C07280=1094.972,417.222,400.209,178.802,23.550,153.433
C07281=1094.966,417.006,400.244,178.799,23.542,153.431
C07282=1094.960,416.791,400.280,178.797,23.534,153.429
C07283=1094.956,416.575,400.315,178.794,23.526,153.428
C07284=1094.950,416.359,400.351,178.792,23.518,153.426
C07285=1094.945,416.144,400.387,178.789,23.510,153.424
C07286=1094.938,415.897,400.427,178.786,23.501,153.423
C07287=1094.933,415.650,400.467,178.783,23.492,153.421
C07288=1094.926,415.404,400.508,178.780,23.483,153.419
C07289=1094.920,415.157,400.548,178.778,23.475,153.417
C07290=1094.914,414.910,400.589,178.776,23.466,153.415
C07291=1094.908,414.664,400.629,178.772,23.457,153.414
C07292=1094.902,414.417,400.669,178.770,23.448,153.412
C07293=1094.896,414.170,400.710,178.767,23.439,153.410
C07294=1094.890,413.923,400.749,178.764,23.431,153.408
C07295=1094.883,413.677,400.789,178.762,23.422,153.407
C07296=1094.877,413.430,400.829,178.758,23.414,153.405
C07297=1094.871,413.184,400.870,178.756,23.405,153.403
C07298=1094.865,412.937,400.910,178.753,23.396,153.401
C07299=1094.859,412.690,400.950,178.750,23.387,153.400
C07300=1094.853,412.443,400.990,178.747,23.379,153.398
C07301=1094.847,412.197,401.030,178.744,23.371,153.396
C07302=1094.841,411.951,401.070,178.741,23.362,153.395
C07303=1094.835,411.704,401.110,178.738,23.353,153.393
C07304=1094.829,411.457,401.150,178.736,23.345,153.391
C07305=1094.823,411.210,401.191,178.733,23.337,153.390
C07306=1094.816,410.955,401.232,178.730,23.328,153.388
C07307=1094.810,410.698,401.273,178.727,23.319,153.386
C07308=1094.804,410.442,401.314,178.724,23.311,153.384
C07309=1094.798,410.186,401.356,178.721,23.302,153.383
C07310=1094.791,409.939,401.396,178.719,23.294,153.381
C07311=1094.785,409.692,401.435,178.716,23.286,153.379
C07312=1094.780,409.446,401.476,178.713,23.277,153.378
C07313=1094.774,409.199,401.515,178.711,23.269,153.376
C07314=1094.768,408.952,401.555,178.708,23.261,153.374
C07315=1094.762,408.705,401.595,178.705,23.253,153.373
C07316=1094.755,408.459,401.635,178.702,23.245,153.371
C07317=1094.750,408.212,401.674,178.699,23.237,153.370
C07318=1094.744,407.965,401.713,178.696,23.228,153.368
C07319=1094.738,407.718,401.754,178.694,23.220,153.366
C07320=1094.732,407.471,401.793,178.691,23.212,153.365
C07321=1094.727,407.225,401.833,178.688,23.205,153.363
C07322=1094.720,406.978,401.873,178.685,23.196,153.362
C07323=1094.714,406.731,401.912,178.682,23.188,153.360
C07324=1094.708,406.484,401.952,178.680,23.180,153.359
C07325=1094.703,406.237,401.991,178.677,23.172,153.357
C07326=1094.695,405.991,402.030,178.674,23.164,153.356
C07327=1094.689,405.744,402.070,178.671,23.156,153.354
C07328=1094.683,405.497,402.109,178.669,23.149,153.353
C07329=1094.678,405.250,402.148,178.666,23.141,153.351
C07330=1094.672,405.003,402.188,178.663,23.133,153.349
C07331=1094.666,404.756,402.227,178.660,23.126,153.348
C07332=1094.660,404.510,402.266,178.657,23.118,153.347
C07333=1094.654,404.263,402.305,178.655,23.110,153.345
C07334=1094.648,404.015,402.345,178.651,23.102,153.344
C07335=1094.642,403.769,402.383,178.649,23.095,153.342
C07336=1094.636,403.522,402.423,178.646,23.087,153.341
C07337=1094.630,403.275,402.462,178.643,23.080,153.339
C07338=1094.624,403.029,402.501,178.640,23.072,153.338
C07339=1094.617,402.782,402.540,178.638,23.064,153.336
C07340=1094.611,402.535,402.580,178.635,23.057,153.335
C07341=1094.606,402.288,402.619,178.632,23.049,153.333
C07342=1094.600,402.041,402.658,178.630,23.042,153.332
C07343=1094.593,401.794,402.697,178.626,23.034,153.331
C07344=1094.588,401.548,402.736,178.624,23.027,153.329
C07345=1094.581,401.301,402.775,178.620,23.019,153.328
C07346=1094.576,401.054,402.814,178.618,23.012,153.326
C07347=1094.569,400.807,402.853,178.615,23.005,153.325
C07348=1094.564,400.560,402.892,178.612,22.997,153.324
C07349=1094.558,400.313,402.931,178.610,22.990,153.322
C07350=1094.551,400.066,402.969,178.607,22.982,153.321
C07351=1094.546,399.819,403.008,178.604,22.975,153.319
C07352=1094.540,399.572,403.048,178.601,22.968,153.318
C07353=1094.534,399.326,403.085,178.598,22.961,153.317
C07354=1094.528,399.078,403.125,178.596,22.954,153.315
C07355=1094.522,398.832,403.163,178.592,22.946,153.314
C07356=1094.516,398.584,403.202,178.590,22.939,153.313
C07357=1094.510,398.338,403.241,178.587,22.932,153.311
C07358=1094.504,398.118,403.275,178.585,22.926,153.310
C07359=1094.499,397.898,403.309,178.582,22.919,153.309
C07360=1094.493,397.677,403.344,178.579,22.913,153.308
C07361=1094.489,397.458,403.379,178.577,22.907,153.306
C07362=1094.483,397.237,403.414,178.575,22.900,153.305
C07363=1094.478,397.017,403.448,178.572,22.894,153.304
C07364=1094.473,396.798,403.482,178.569,22.888,153.303
C07365=1094.468,396.577,403.516,178.567,22.882,153.302
C07366=1094.461,396.331,403.555,178.564,22.874,153.301
C07367=1094.455,396.083,403.593,178.561,22.868,153.299
C07368=1094.450,395.836,403.631,178.559,22.861,153.298
C07369=1094.443,395.590,403.670,178.556,22.854,153.297
C07370=1094.438,395.343,403.708,178.553,22.847,153.295
C07371=1094.432,395.096,403.746,178.550,22.840,153.294
C07372=1094.426,394.849,403.786,178.548,22.833,153.293
C07373=1094.420,394.602,403.823,178.544,22.826,153.292
C07374=1094.414,394.355,403.861,178.541,22.819,153.290
C07375=1094.408,394.108,403.901,178.539,22.813,153.289
C07376=1094.402,393.861,403.938,178.536,22.806,153.288
C07377=1094.396,393.615,403.976,178.533,22.799,153.287
C07378=1094.390,393.367,404.015,178.530,22.792,153.285
C07379=1094.384,393.121,404.053,178.527,22.786,153.284
C07380=1094.378,392.874,404.091,178.525,22.779,153.283
C07381=1094.372,392.626,404.129,178.521,22.772,153.282
C07382=1094.366,392.379,404.167,178.519,22.765,153.281
C07383=1094.361,392.133,404.205,178.516,22.759,153.279
C07384=1094.354,391.885,404.243,178.513,22.752,153.278
C07385=1094.348,391.638,404.281,178.511,22.746,153.277
C07386=1094.342,391.392,404.319,178.507,22.739,153.276
C07387=1094.336,391.144,404.357,178.504,22.732,153.275
C07388=1094.330,390.898,404.395,178.502,22.726,153.274
C07389=1094.324,390.651,404.434,178.499,22.720,153.272
C07390=1094.318,390.403,404.471,178.496,22.713,153.271
C07391=1094.312,390.156,404.509,178.493,22.706,153.270
C07392=1094.306,389.910,404.547,178.490,22.700,153.269
C07393=1094.300,389.663,404.584,178.487,22.694,153.268
C07394=1094.295,389.416,404.622,178.485,22.687,153.267
C07395=1094.288,389.169,404.660,178.482,22.681,153.266
C07396=1094.282,388.922,404.698,178.478,22.674,153.265
C07397=1094.276,388.675,404.736,178.475,22.668,153.263
C07398=1094.270,388.428,404.774,178.473,22.662,153.262
C07399=1094.264,388.182,404.811,178.470,22.655,153.261
C07400=1094.258,387.934,404.849,178.467,22.649,153.260
C07401=1094.252,387.687,404.887,178.464,22.643,153.259
C07402=1094.246,387.440,404.924,178.461,22.636,153.258
C07403=1094.240,387.193,404.962,178.458,22.630,153.257
C07404=1094.235,386.947,405.000,178.455,22.624,153.256
C07405=1094.229,386.699,405.037,178.452,22.617,153.254
C07406=1094.223,386.453,405.075,178.450,22.611,153.253
C07407=1094.217,386.205,405.113,178.447,22.605,153.252
C07408=1094.211,385.958,405.150,178.444,22.599,153.251
C07409=1094.205,385.711,405.188,178.441,22.593,153.250
C07410=1094.199,385.464,405.225,178.438,22.586,153.249
C07411=1094.194,385.217,405.262,178.435,22.580,153.248
C07412=1094.188,384.970,405.300,178.432,22.574,153.247
C07413=1094.182,384.723,405.337,178.429,22.568,153.246
C07414=1094.177,384.509,405.370,178.427,22.563,153.245
C07415=1094.172,384.296,405.402,178.424,22.557,153.244
C07416=1094.166,384.082,405.434,178.422,22.552,153.243
C07417=1094.161,383.869,405.466,178.420,22.547,153.242
C07418=1094.156,383.655,405.498,178.417,22.542,153.242
C07419=1094.151,383.441,405.531,178.415,22.536,153.240
C07420=1094.146,383.228,405.563,178.411,22.531,153.240
C07421=1094.142,383.014,405.595,178.409,22.525,153.239
C07422=1094.136,382.767,405.633,178.406,22.519,153.238
C07423=1094.130,382.520,405.670,178.404,22.514,153.237
C07424=1094.124,382.273,405.706,178.401,22.508,153.236
C07425=1094.118,382.026,405.744,178.398,22.502,153.235
C07426=1094.112,381.778,405.782,178.395,22.496,153.234
C07427=1094.105,381.531,405.818,178.392,22.490,153.233
C07428=1094.099,381.284,405.856,178.389,22.485,153.232
C07429=1094.094,381.037,405.893,178.386,22.479,153.231
C07430=1094.087,380.790,405.929,178.383,22.473,153.230
C07431=1094.081,380.543,405.967,178.380,22.467,153.229
C07432=1094.076,380.296,406.004,178.377,22.461,153.228
C07433=1094.070,380.049,406.041,178.374,22.455,153.227
C07434=1094.064,379.801,406.078,178.371,22.450,153.226
C07435=1094.058,379.554,406.115,178.369,22.444,153.225
C07436=1094.052,379.308,406.151,178.366,22.438,153.224
C07437=1094.047,379.061,406.188,178.363,22.432,153.223
C07438=1094.040,378.814,406.225,178.360,22.427,153.222
C07439=1094.035,378.567,406.262,178.357,22.421,153.221
C07440=1094.029,378.319,406.299,178.354,22.415,153.220
C07441=1094.023,378.072,406.335,178.351,22.409,153.220
C07442=1094.017,377.825,406.372,178.348,22.403,153.218
C07443=1094.011,377.578,406.409,178.345,22.398,153.218
C07444=1094.005,377.330,406.446,178.342,22.392,153.217
C07445=1093.999,377.083,406.482,178.339,22.386,153.216
C07446=1093.993,376.836,406.519,178.336,22.381,153.215
C07447=1093.988,376.589,406.556,178.333,22.375,153.214
C07448=1093.982,376.342,406.593,178.330,22.370,153.213
C07449=1093.976,376.095,406.630,178.327,22.364,153.212
C07450=1093.970,375.848,406.666,178.324,22.358,153.211
C07451=1093.965,375.600,406.703,178.321,22.353,153.210
C07452=1093.958,375.353,406.739,178.318,22.347,153.209
C07453=1093.953,375.105,406.776,178.315,22.342,153.209
C07454=1093.947,374.859,406.812,178.312,22.336,153.208
C07455=1093.942,374.612,406.849,178.309,22.331,153.207
C07456=1093.935,374.365,406.885,178.307,22.325,153.206
C07457=1093.930,374.117,406.922,178.304,22.320,153.205
C07458=1093.924,373.870,406.958,178.301,22.314,153.204
C07459=1093.917,373.623,406.995,178.298,22.309,153.203
C07460=1093.912,373.376,407.031,178.295,22.304,153.203
C07461=1093.906,373.129,407.068,178.292,22.298,153.202
C07462=1093.900,372.881,407.103,178.289,22.293,153.201
C07463=1093.894,372.634,407.140,178.285,22.287,153.200
C07464=1093.888,372.387,407.177,178.282,22.282,153.199
C07465=1093.883,372.140,407.212,178.280,22.277,153.198
C07466=1093.876,371.893,407.249,178.277,22.272,153.198
C07467=1093.871,371.645,407.285,178.274,22.266,153.197
C07468=1093.865,371.398,407.322,178.271,22.261,153.196
C07469=1093.858,371.151,407.358,178.268,22.255,153.195
C07470=1093.849,370.751,407.416,178.263,22.247,153.194
C07471=1093.840,370.351,407.474,178.258,22.238,153.192
C07472=1093.830,369.951,407.533,178.254,22.230,153.191
C07473=1093.821,369.552,407.591,178.249,22.222,153.190
C07474=1093.815,369.304,407.627,178.246,22.217,153.189
C07475=1093.808,369.057,407.663,178.243,22.211,153.188
C07476=1093.804,368.810,407.699,178.240,22.206,153.187
C07477=1093.798,368.562,407.735,178.236,22.201,153.187
C07478=1093.791,368.315,407.771,178.234,22.196,153.186
C07479=1093.785,368.067,407.807,178.231,22.190,153.185
C07480=1093.780,367.820,407.843,178.228,22.185,153.184
C07481=1093.774,367.573,407.880,178.225,22.180,153.184
C07482=1093.769,367.326,407.915,178.222,22.175,153.183
C07483=1093.763,367.078,407.951,178.218,22.170,153.182
C07484=1093.757,366.831,407.986,178.216,22.165,153.181
C07485=1093.751,366.584,408.023,178.213,22.160,153.180
C07486=1093.745,366.337,408.058,178.210,22.155,153.180
C07487=1093.739,366.089,408.094,178.207,22.150,153.179
C07488=1093.734,365.842,408.129,178.204,22.144,153.178
C07489=1093.728,365.594,408.165,178.201,22.140,153.177
C07490=1093.722,365.347,408.201,178.198,22.135,153.177
C07491=1093.716,365.100,408.237,178.195,22.130,153.176
C07492=1093.710,364.853,408.273,178.192,22.125,153.175
C07493=1093.704,364.606,408.308,178.189,22.120,153.175
C07494=1093.698,364.358,408.344,178.186,22.115,153.174
C07495=1093.692,364.110,408.379,178.183,22.110,153.173
C07496=1093.687,363.863,408.415,178.180,22.105,153.172
C07497=1093.681,363.616,408.451,178.177,22.101,153.172
C07498=1093.675,363.369,408.486,178.174,22.095,153.171
C07499=1093.669,363.121,408.522,178.171,22.090,153.170
C07500=1093.663,362.873,408.557,178.168,22.085,153.170
C07501=1093.658,362.626,408.593,178.165,22.081,153.169
C07502=1093.652,362.379,408.628,178.162,22.076,153.168
C07503=1093.647,362.132,408.664,178.159,22.071,153.168
C07504=1093.640,361.884,408.699,178.156,22.066,153.167
C07505=1093.635,361.637,408.734,178.153,22.061,153.166
C07506=1093.629,361.389,408.769,178.150,22.057,153.166
C07507=1093.623,361.141,408.805,178.147,22.052,153.165
C07508=1093.617,360.894,408.840,178.143,22.047,153.164
C07509=1093.611,360.647,408.876,178.141,22.042,153.163
C07510=1093.605,360.400,408.911,178.138,22.038,153.163
C07511=1093.599,360.152,408.946,178.135,22.032,153.162
C07512=1093.594,359.905,408.981,178.132,22.028,153.161
C07513=1093.588,359.657,409.017,178.129,22.024,153.161
C07514=1093.583,359.409,409.052,178.126,22.018,153.160
C07515=1093.576,359.162,409.087,178.122,22.014,153.160
C07516=1093.570,358.915,409.122,178.120,22.009,153.159
C07517=1093.564,358.667,409.158,178.117,22.004,153.158
C07518=1093.559,358.420,409.192,178.113,22.000,153.158
C07519=1093.553,358.172,409.228,178.111,21.995,153.157
C07520=1093.547,357.925,409.262,178.107,21.991,153.156
C07521=1093.541,357.678,409.297,178.104,21.986,153.156
C07522=1093.532,357.293,409.351,178.100,21.979,153.155
C07523=1093.523,356.908,409.407,178.095,21.972,153.154
C07524=1093.514,356.524,409.461,178.091,21.965,153.153
C07525=1093.505,356.139,409.515,178.085,21.957,153.152
C07526=1093.499,355.892,409.550,178.083,21.953,153.151
C07527=1093.493,355.644,409.585,178.080,21.948,153.151
C07528=1093.488,355.397,409.620,178.076,21.943,153.150
C07529=1093.482,355.150,409.654,178.074,21.939,153.149
C07530=1093.476,354.902,409.690,178.070,21.934,153.149
C07531=1093.470,354.655,409.724,178.067,21.930,153.148
C07532=1093.464,354.406,409.759,178.065,21.926,153.147
C07533=1093.459,354.160,409.794,178.061,21.921,153.147
C07534=1093.453,353.912,409.828,178.059,21.917,153.146
C07535=1093.447,353.664,409.863,178.055,21.912,153.146
C07536=1093.441,353.417,409.898,178.052,21.908,153.145
C07537=1093.436,353.170,409.933,178.049,21.903,153.145
C07538=1093.430,352.922,409.967,178.046,21.899,153.144
C07539=1093.425,352.674,410.002,178.043,21.894,153.143
C07540=1093.418,352.427,410.037,178.040,21.890,153.143
C07541=1093.412,352.179,410.071,178.037,21.886,153.142
C07542=1093.407,351.932,410.106,178.034,21.881,153.142
C07543=1093.400,351.684,410.140,178.031,21.877,153.141
C07544=1093.395,351.436,410.175,178.027,21.872,153.141
C07545=1093.389,351.190,410.209,178.025,21.868,153.140
C07546=1093.383,350.942,410.244,178.021,21.864,153.140
C07547=1093.377,350.694,410.279,178.019,21.860,153.139
C07548=1093.372,350.447,410.313,178.016,21.855,153.138
C07549=1093.367,350.199,410.347,178.012,21.851,153.138
C07550=1093.360,349.951,410.382,178.010,21.846,153.137
C07551=1093.354,349.704,410.416,178.006,21.842,153.137
C07552=1093.349,349.456,410.450,178.004,21.838,153.136
C07553=1093.343,349.208,410.485,178.000,21.834,153.136
C07554=1093.337,348.961,410.519,177.998,21.829,153.135
C07555=1093.332,348.713,410.553,177.994,21.825,153.135
C07556=1093.326,348.466,410.588,177.992,21.821,153.134
C07557=1093.319,348.218,410.622,177.988,21.817,153.134
C07558=1093.313,347.971,410.656,177.985,21.812,153.133
C07559=1093.308,347.723,410.691,177.982,21.808,153.133
C07560=1093.302,347.476,410.725,177.979,21.804,153.132
C07561=1093.296,347.228,410.759,177.976,21.800,153.131
C07562=1093.291,346.980,410.794,177.973,21.795,153.131
C07563=1093.285,346.733,410.827,177.970,21.791,153.130
C07564=1093.279,346.485,410.861,177.967,21.787,153.130
C07565=1093.274,346.238,410.895,177.964,21.783,153.129
C07566=1093.268,345.991,410.929,177.961,21.778,153.129
C07567=1093.262,345.742,410.964,177.958,21.775,153.128
C07568=1093.256,345.494,410.998,177.955,21.770,153.128
C07569=1093.251,345.247,411.032,177.951,21.766,153.127
C07570=1093.245,345.000,411.066,177.949,21.762,153.127
C07571=1093.239,344.753,411.100,177.945,21.758,153.126
C07572=1093.233,344.504,411.134,177.942,21.754,153.126
C07573=1093.228,344.256,411.168,177.939,21.750,153.125
C07574=1093.219,343.874,411.220,177.934,21.743,153.125
C07575=1093.209,343.492,411.273,177.930,21.737,153.124
C07576=1093.201,343.110,411.324,177.925,21.731,153.123
C07577=1093.191,342.728,411.377,177.921,21.725,153.123
C07578=1093.186,342.481,411.411,177.917,21.721,153.122
C07579=1093.180,342.233,411.445,177.914,21.717,153.122
C07580=1093.174,341.985,411.478,177.911,21.713,153.121
C07581=1093.168,341.738,411.512,177.908,21.709,153.121
C07582=1093.163,341.490,411.545,177.905,21.705,153.120
C07583=1093.157,341.243,411.579,177.902,21.701,153.120
C07584=1093.151,340.995,411.613,177.899,21.697,153.119
C07585=1093.146,340.748,411.647,177.896,21.693,153.119
C07586=1093.140,340.500,411.680,177.892,21.688,153.118
C07587=1093.134,340.252,411.715,177.890,21.685,153.118
C07588=1093.128,340.004,411.748,177.886,21.680,153.117
C07589=1093.122,339.756,411.781,177.883,21.677,153.117
C07590=1093.117,339.509,411.815,177.881,21.673,153.117
C07591=1093.111,339.261,411.849,177.877,21.669,153.116
C07592=1093.106,339.013,411.882,177.875,21.665,153.116
C07593=1093.100,338.766,411.916,177.871,21.661,153.115
C07594=1093.094,338.518,411.949,177.868,21.657,153.115
C07595=1093.088,338.270,411.982,177.865,21.653,153.114
C07596=1093.082,338.023,412.016,177.862,21.650,153.114
C07597=1093.076,337.775,412.050,177.859,21.646,153.113
C07598=1093.071,337.527,412.083,177.856,21.642,153.113
C07599=1093.065,337.279,412.116,177.853,21.638,153.113
C07600=1093.059,337.032,412.149,177.850,21.634,153.112
C07601=1093.053,336.784,412.183,177.847,21.630,153.112
C07602=1093.048,336.536,412.216,177.843,21.626,153.111
C07603=1093.042,336.288,412.250,177.840,21.623,153.111
C07604=1093.036,336.041,412.282,177.838,21.619,153.111
C07605=1093.030,335.793,412.316,177.834,21.615,153.110
C07606=1093.025,335.545,412.349,177.831,21.611,153.110
C07607=1093.019,335.298,412.383,177.828,21.607,153.109
C07608=1093.012,335.050,412.416,177.825,21.604,153.109
C07609=1093.007,334.802,412.449,177.822,21.600,153.109
C07610=1093.001,334.554,412.483,177.819,21.596,153.108
C07611=1092.996,334.306,412.516,177.816,21.592,153.108
C07612=1092.989,334.059,412.549,177.812,21.589,153.107
C07613=1092.984,333.811,412.582,177.810,21.585,153.107
C07614=1092.979,333.564,412.615,177.807,21.581,153.107
C07615=1092.973,333.316,412.648,177.803,21.577,153.106
C07616=1092.967,333.068,412.681,177.801,21.574,153.106
C07617=1092.962,332.820,412.714,177.798,21.570,153.105
C07618=1092.955,332.573,412.747,177.794,21.566,153.105
C07619=1092.950,332.324,412.780,177.792,21.562,153.105
C07620=1092.944,332.076,412.813,177.788,21.559,153.104
C07621=1092.938,331.829,412.846,177.785,21.555,153.104
C07622=1092.933,331.581,412.879,177.782,21.551,153.103
C07623=1092.926,331.333,412.912,177.779,21.548,153.103
C07624=1092.920,331.086,412.945,177.776,21.544,153.103
C07625=1092.915,330.838,412.978,177.773,21.541,153.103
C07626=1092.905,330.450,413.029,177.768,21.535,153.102
C07627=1092.896,330.062,413.080,177.763,21.529,153.101
C07628=1092.887,329.674,413.132,177.758,21.524,153.101
C07629=1092.878,329.286,413.183,177.754,21.518,153.100
C07630=1092.872,329.039,413.215,177.750,21.515,153.100
C07631=1092.867,328.790,413.248,177.747,21.511,153.100
C07632=1092.861,328.542,413.281,177.745,21.508,153.099
C07633=1092.854,328.295,413.314,177.741,21.504,153.099
C07634=1092.849,328.046,413.346,177.738,21.501,153.099
C07635=1092.843,327.799,413.379,177.735,21.497,153.098
C07636=1092.837,327.551,413.411,177.732,21.493,153.098
C07637=1092.832,327.303,413.444,177.729,21.490,153.098
C07638=1092.826,327.056,413.477,177.726,21.487,153.097
C07639=1092.820,326.808,413.509,177.722,21.482,153.097
C07640=1092.815,326.560,413.542,177.720,21.479,153.097
C07641=1092.809,326.312,413.574,177.717,21.476,153.096
C07642=1092.802,326.065,413.606,177.714,21.472,153.096
C07643=1092.797,325.816,413.639,177.710,21.469,153.096
C07644=1092.791,325.569,413.671,177.707,21.465,153.095
C07645=1092.785,325.321,413.703,177.705,21.462,153.095
C07646=1092.780,325.073,413.737,177.701,21.458,153.095
C07647=1092.774,324.825,413.769,177.698,21.455,153.094
C07648=1092.768,324.578,413.801,177.695,21.452,153.094
C07649=1092.762,324.330,413.833,177.692,21.448,153.094
C07650=1092.757,324.081,413.866,177.688,21.445,153.093
C07651=1092.751,323.834,413.899,177.686,21.441,153.093
C07652=1092.745,323.586,413.930,177.683,21.438,153.093
C07653=1092.739,323.338,413.963,177.680,21.435,153.092
C07654=1092.734,323.090,413.996,177.676,21.431,153.092
C07655=1092.728,322.842,414.027,177.673,21.427,153.092
C07656=1092.722,322.594,414.059,177.671,21.424,153.091
C07657=1092.716,322.347,414.092,177.668,21.421,153.091
C07658=1092.711,322.099,414.124,177.664,21.417,153.091
C07659=1092.705,321.851,414.156,177.661,21.414,153.091
C07660=1092.700,321.604,414.189,177.658,21.410,153.090
C07661=1092.694,321.355,414.221,177.655,21.407,153.090
C07662=1092.688,321.107,414.253,177.652,21.403,153.090
C07663=1092.682,320.860,414.284,177.649,21.400,153.089
C07664=1092.677,320.611,414.317,177.646,21.397,153.089
C07665=1092.671,320.364,414.350,177.643,21.394,153.089
C07666=1092.665,320.116,414.381,177.639,21.390,153.089
C07667=1092.659,319.868,414.413,177.637,21.386,153.088
C07668=1092.654,319.620,414.445,177.634,21.383,153.088
C07669=1092.648,319.372,414.477,177.631,21.380,153.088
C07670=1092.643,319.124,414.509,177.627,21.376,153.087
C07671=1092.637,318.876,414.541,177.624,21.373,153.087
C07672=1092.632,318.629,414.573,177.621,21.370,153.087
C07673=1092.626,318.380,414.605,177.619,21.366,153.086
C07674=1092.621,318.133,414.637,177.616,21.363,153.086
C07675=1092.615,317.885,414.669,177.612,21.360,153.086
C07676=1092.609,317.637,414.700,177.609,21.356,153.086
C07677=1092.603,317.389,414.733,177.606,21.353,153.085
C07678=1092.595,316.994,414.784,177.601,21.347,153.085
C07679=1092.586,316.599,414.835,177.597,21.343,153.084
C07680=1092.577,316.204,414.885,177.592,21.337,153.084
C07681=1092.568,315.809,414.935,177.587,21.332,153.083
C07682=1092.563,315.562,414.968,177.584,21.328,153.083
C07683=1092.557,315.313,415.000,177.581,21.325,153.083
C07684=1092.552,315.066,415.031,177.578,21.322,153.083
C07685=1092.545,314.818,415.063,177.574,21.319,153.082
C07686=1092.540,314.570,415.094,177.571,21.315,153.082
C07687=1092.534,314.322,415.126,177.568,21.312,153.082
C07688=1092.527,314.074,415.157,177.565,21.309,153.082
C07689=1092.522,313.826,415.189,177.562,21.306,153.081
C07690=1092.516,313.578,415.221,177.559,21.303,153.081
C07691=1092.511,313.330,415.252,177.556,21.299,153.081
C07692=1092.504,313.082,415.283,177.553,21.296,153.081
C07693=1092.499,312.834,415.315,177.550,21.293,153.081
C07694=1092.493,312.586,415.347,177.547,21.290,153.080
C07695=1092.487,312.338,415.377,177.544,21.287,153.080
C07696=1092.481,312.091,415.409,177.541,21.284,153.080
C07697=1092.475,311.843,415.441,177.537,21.281,153.080
C07698=1092.470,311.595,415.471,177.534,21.277,153.079
C07699=1092.464,311.347,415.503,177.531,21.275,153.079
C07700=1092.458,311.099,415.534,177.528,21.272,153.079
C07701=1092.452,310.851,415.566,177.525,21.268,153.079
C07702=1092.446,310.603,415.597,177.522,21.265,153.078
C07703=1092.441,310.355,415.628,177.519,21.262,153.078
C07704=1092.435,310.107,415.660,177.515,21.259,153.078
C07705=1092.429,309.859,415.691,177.513,21.256,153.078
C07706=1092.423,309.611,415.722,177.509,21.253,153.078
C07707=1092.418,309.363,415.753,177.506,21.250,153.077
C07708=1092.412,309.115,415.785,177.503,21.247,153.077
C07709=1092.406,308.867,415.815,177.501,21.244,153.077
C07710=1092.400,308.619,415.847,177.498,21.241,153.077
C07711=1092.395,308.372,415.877,177.494,21.237,153.077
C07712=1092.389,308.123,415.909,177.491,21.234,153.076
C07713=1092.383,307.875,415.940,177.488,21.231,153.076
C07714=1092.377,307.628,415.972,177.485,21.228,153.076
C07715=1092.372,307.379,416.003,177.482,21.225,153.076
C07716=1092.366,307.132,416.034,177.479,21.222,153.075
C07717=1092.361,306.884,416.065,177.476,21.219,153.075
C07718=1092.354,306.635,416.096,177.472,21.216,153.075
C07719=1092.349,306.388,416.127,177.469,21.213,153.075
C07720=1092.343,306.140,416.158,177.466,21.210,153.075
C07721=1092.338,305.892,416.189,177.463,21.207,153.074
C07722=1092.331,305.644,416.220,177.460,21.204,153.074
C07723=1092.326,305.396,416.251,177.457,21.201,153.074
C07724=1092.320,305.148,416.281,177.454,21.198,153.074
C07725=1092.315,304.900,416.312,177.451,21.195,153.074
C07726=1092.309,304.653,416.343,177.447,21.191,153.073
C07727=1092.303,304.404,416.375,177.444,21.188,153.073
C07728=1092.298,304.156,416.405,177.441,21.185,153.073
C07729=1092.292,303.908,416.436,177.438,21.183,153.073
C07730=1092.283,303.516,416.485,177.434,21.178,153.072
C07731=1092.274,303.123,416.533,177.429,21.173,153.072
C07732=1092.265,302.732,416.582,177.424,21.168,153.072
C07733=1092.257,302.339,416.631,177.419,21.163,153.072
C07734=1092.251,302.091,416.661,177.416,21.160,153.071
C07735=1092.246,301.843,416.692,177.413,21.157,153.071
C07736=1092.240,301.595,416.723,177.410,21.154,153.071
C07737=1092.234,301.347,416.753,177.407,21.151,153.071
C07738=1092.229,301.099,416.784,177.404,21.149,153.071
C07739=1092.223,300.851,416.814,177.401,21.146,153.070
C07740=1092.218,300.603,416.845,177.398,21.143,153.070
C07741=1092.212,300.355,416.876,177.395,21.140,153.070
C07742=1092.206,300.107,416.906,177.391,21.136,153.070
C07743=1092.201,299.858,416.937,177.388,21.133,153.070
C07744=1092.195,299.611,416.968,177.385,21.130,153.069
C07745=1092.189,299.363,416.998,177.382,21.127,153.069
C07746=1092.184,299.115,417.029,177.379,21.124,153.069
C07747=1092.178,298.867,417.059,177.376,21.121,153.069
C07748=1092.173,298.619,417.090,177.373,21.118,153.069
C07749=1092.167,298.371,417.121,177.370,21.115,153.068
C07750=1092.161,298.123,417.151,177.367,21.113,153.068
C07751=1092.156,297.875,417.181,177.364,21.110,153.068
C07752=1092.151,297.627,417.211,177.361,21.107,153.068
C07753=1092.145,297.379,417.242,177.358,21.104,153.068
C07754=1092.139,297.131,417.272,177.355,21.101,153.068
C07755=1092.133,296.883,417.303,177.352,21.098,153.068
C07756=1092.127,296.634,417.333,177.349,21.096,153.067
C07757=1092.121,296.386,417.363,177.346,21.093,153.067
C07758=1092.116,296.138,417.393,177.343,21.090,153.067
C07759=1092.111,295.890,417.424,177.340,21.087,153.067
C07760=1092.105,295.642,417.454,177.337,21.084,153.067
C07761=1092.099,295.394,417.484,177.334,21.081,153.067
C07762=1092.093,295.146,417.515,177.331,21.078,153.066
C07763=1092.088,294.898,417.544,177.328,21.076,153.066
C07764=1092.082,294.650,417.575,177.325,21.073,153.066
C07765=1092.076,294.402,417.605,177.321,21.070,153.066
C07766=1092.071,294.154,417.634,177.318,21.067,153.066
C07767=1092.065,293.906,417.665,177.315,21.064,153.066
C07768=1092.059,293.658,417.695,177.312,21.061,153.065
C07769=1092.054,293.409,417.725,177.309,21.058,153.065
C07770=1092.048,293.162,417.755,177.305,21.056,153.065
C07771=1092.042,292.913,417.785,177.302,21.053,153.065
C07772=1092.036,292.665,417.815,177.299,21.050,153.065
C07773=1092.031,292.417,417.845,177.296,21.047,153.065
C07774=1092.025,292.169,417.875,177.293,21.044,153.065
C07775=1092.020,291.921,417.905,177.290,21.041,153.065
C07776=1092.014,291.673,417.935,177.287,21.038,153.064
C07777=1092.008,291.424,417.965,177.284,21.036,153.064
C07778=1092.003,291.177,417.995,177.281,21.033,153.064
C07779=1091.997,290.928,418.025,177.278,21.030,153.064
C07780=1091.991,290.680,418.054,177.275,21.027,153.064
C07781=1091.985,290.432,418.084,177.272,21.025,153.064
C07782=1091.977,290.054,418.130,177.267,21.020,153.063
C07783=1091.969,289.675,418.175,177.262,21.016,153.063
C07784=1091.960,289.297,418.221,177.258,21.012,153.063
C07785=1091.951,288.919,418.266,177.253,21.008,153.063
C07786=1091.945,288.671,418.295,177.250,21.005,153.063
C07787=1091.939,288.423,418.325,177.247,21.003,153.063
C07788=1091.934,288.175,418.355,177.244,21.000,153.063
C07789=1091.928,287.926,418.385,177.241,20.997,153.062
C07790=1091.922,287.678,418.414,177.238,20.994,153.062
C07791=1091.917,287.431,418.444,177.235,20.992,153.062
C07792=1091.911,287.182,418.473,177.232,20.989,153.062
C07793=1091.906,286.934,418.503,177.229,20.986,153.062
C07794=1091.899,286.686,418.532,177.226,20.984,153.062
C07795=1091.894,286.437,418.562,177.223,20.981,153.062
C07796=1091.888,286.190,418.592,177.220,20.979,153.062
C07797=1091.882,285.941,418.621,177.217,20.976,153.061
C07798=1091.876,285.693,418.651,177.214,20.973,153.061
C07799=1091.871,285.445,418.680,177.211,20.970,153.061
C07800=1091.866,285.197,418.710,177.208,20.968,153.061
C07801=1091.860,284.949,418.739,177.204,20.965,153.061
C07802=1091.854,284.700,418.768,177.202,20.962,153.061
C07803=1091.849,284.452,418.798,177.198,20.960,153.061
C07804=1091.842,284.204,418.827,177.195,20.957,153.061
C07805=1091.837,283.956,418.856,177.192,20.954,153.061
C07806=1091.832,283.707,418.886,177.189,20.951,153.060
C07807=1091.826,283.459,418.915,177.186,20.948,153.060
C07808=1091.820,283.211,418.945,177.183,20.946,153.060
C07809=1091.815,282.963,418.974,177.180,20.943,153.060
C07810=1091.809,282.715,419.003,177.177,20.941,153.060
C07811=1091.803,282.467,419.032,177.175,20.938,153.060
C07812=1091.798,282.218,419.062,177.171,20.936,153.060
C07813=1091.792,281.971,419.091,177.168,20.933,153.060
C07814=1091.787,281.722,419.120,177.165,20.930,153.060
C07815=1091.780,281.474,419.149,177.162,20.927,153.059
C07816=1091.775,281.226,419.179,177.159,20.925,153.059
C07817=1091.770,280.978,419.208,177.156,20.922,153.059
C07818=1091.764,280.729,419.237,177.153,20.919,153.059
C07819=1091.758,280.481,419.266,177.149,20.917,153.059
C07820=1091.752,280.233,419.295,177.146,20.914,153.059
C07821=1091.747,279.985,419.324,177.143,20.912,153.059
C07822=1091.741,279.737,419.354,177.140,20.909,153.059
C07823=1091.735,279.488,419.382,177.138,20.907,153.059
C07824=1091.730,279.240,419.412,177.135,20.904,153.059
C07825=1091.724,278.992,419.440,177.132,20.901,153.058
C07826=1091.719,278.744,419.470,177.128,20.899,153.058
C07827=1091.713,278.495,419.498,177.125,20.896,153.058
C07828=1091.707,278.246,419.528,177.122,20.893,153.058
C07829=1091.701,277.999,419.557,177.119,20.891,153.058
C07830=1091.696,277.750,419.585,177.116,20.888,153.058
C07831=1091.690,277.502,419.615,177.113,20.886,153.058
C07832=1091.684,277.254,419.643,177.111,20.883,153.058
C07833=1091.679,277.005,419.672,177.108,20.881,153.058
C07834=1091.670,276.637,419.715,177.103,20.877,153.058
C07835=1091.662,276.268,419.758,177.098,20.873,153.058
C07836=1091.654,275.899,419.801,177.093,20.869,153.057
C07837=1091.646,275.530,419.843,177.090,20.865,153.057
C07838=1091.639,275.282,419.872,177.086,20.863,153.057
C07839=1091.634,275.034,419.900,177.083,20.860,153.057
C07840=1091.628,274.786,419.929,177.080,20.858,153.057
C07841=1091.623,274.537,419.958,177.077,20.855,153.057
C07842=1091.617,274.289,419.987,177.074,20.852,153.057
C07843=1091.611,274.040,420.015,177.071,20.850,153.057
C07844=1091.606,273.793,420.045,177.068,20.847,153.057
C07845=1091.600,273.544,420.073,177.065,20.845,153.057
C07846=1091.594,273.296,420.102,177.062,20.842,153.057
C07847=1091.589,273.048,420.130,177.059,20.840,153.056
C07848=1091.583,272.799,420.160,177.056,20.837,153.056
C07849=1091.578,272.551,420.188,177.053,20.834,153.056
C07850=1091.572,272.302,420.216,177.050,20.832,153.056
C07851=1091.566,272.054,420.245,177.046,20.830,153.056
C07852=1091.560,271.806,420.273,177.044,20.828,153.056
C07853=1091.554,271.558,420.301,177.041,20.825,153.056
C07854=1091.549,271.310,420.330,177.038,20.822,153.056
C07855=1091.543,271.061,420.359,177.035,20.820,153.056
C07856=1091.538,270.813,420.387,177.032,20.817,153.056
C07857=1091.532,270.564,420.415,177.028,20.814,153.056
C07858=1091.527,270.317,420.444,177.026,20.812,153.056
C07859=1091.521,270.068,420.472,177.023,20.810,153.056
C07860=1091.515,269.820,420.500,177.020,20.807,153.056
C07861=1091.510,269.571,420.529,177.017,20.804,153.055
C07862=1091.504,269.323,420.558,177.013,20.802,153.055
C07863=1091.498,269.075,420.586,177.010,20.800,153.055
C07864=1091.492,268.826,420.614,177.008,20.798,153.055
C07865=1091.487,268.578,420.642,177.005,20.795,153.055
C07866=1091.481,268.329,420.671,177.002,20.792,153.055
C07867=1091.476,268.081,420.699,176.998,20.790,153.055
C07868=1091.470,267.832,420.727,176.995,20.787,153.055
C07869=1091.464,267.585,420.756,176.992,20.785,153.055
C07870=1091.458,267.336,420.784,176.990,20.783,153.055
C07871=1091.453,267.088,420.812,176.987,20.780,153.055
C07872=1091.447,266.839,420.840,176.984,20.777,153.055
C07873=1091.442,266.591,420.868,176.980,20.775,153.055
C07874=1091.436,266.343,420.896,176.977,20.772,153.055
C07875=1091.430,266.095,420.924,176.975,20.770,153.055
C07876=1091.425,265.847,420.952,176.972,20.768,153.055
C07877=1091.419,265.598,420.981,176.969,20.765,153.054
C07878=1091.414,265.350,421.009,176.965,20.763,153.054
C07879=1091.408,265.101,421.037,176.962,20.760,153.054
C07880=1091.403,264.853,421.065,176.959,20.758,153.054
C07881=1091.397,264.604,421.093,176.957,20.756,153.054
C07882=1091.391,264.356,421.121,176.954,20.753,153.054
C07883=1091.385,264.108,421.149,176.950,20.750,153.054
C07884=1091.380,263.859,421.176,176.947,20.748,153.054
C07885=1091.374,263.611,421.204,176.944,20.745,153.054
C07886=1091.365,263.245,421.245,176.940,20.742,153.054
C07887=1091.356,262.879,421.286,176.935,20.738,153.054
C07888=1091.348,262.512,421.328,176.931,20.735,153.054
C07889=1091.340,262.146,421.368,176.926,20.732,153.054
C07890=1091.333,261.898,421.396,176.923,20.729,153.054
C07891=1091.328,261.650,421.424,176.921,20.727,153.054
C07892=1091.322,261.401,421.452,176.918,20.725,153.054
C07893=1091.316,261.153,421.479,176.914,20.723,153.054
C07894=1091.311,260.905,421.507,176.911,20.720,153.054
C07895=1091.305,260.656,421.535,176.908,20.717,153.054
C07896=1091.299,260.408,421.563,176.906,20.715,153.054
C07897=1091.293,260.159,421.590,176.903,20.713,153.054
C07898=1091.288,259.911,421.618,176.899,20.710,153.054
C07899=1091.282,259.663,421.646,176.896,20.708,153.054
C07900=1091.276,259.414,421.673,176.894,20.706,153.054
C07901=1091.271,259.166,421.701,176.891,20.703,153.053
C07902=1091.265,258.918,421.729,176.887,20.701,153.053
C07903=1091.259,258.669,421.756,176.884,20.698,153.053
C07904=1091.254,258.421,421.784,176.882,20.696,153.053
C07905=1091.248,258.172,421.811,176.879,20.694,153.053
C07906=1091.242,257.923,421.839,176.875,20.691,153.053
C07907=1091.236,257.676,421.866,176.872,20.689,153.053
C07908=1091.231,257.427,421.894,176.870,20.687,153.053
C07909=1091.225,257.178,421.922,176.867,20.684,153.053
C07910=1091.219,256.930,421.949,176.864,20.682,153.053
C07911=1091.214,256.682,421.977,176.860,20.680,153.053
C07912=1091.208,256.433,422.003,176.858,20.678,153.053
C07913=1091.202,256.185,422.032,176.855,20.675,153.053
C07914=1091.197,255.936,422.059,176.852,20.673,153.053
C07915=1091.192,255.688,422.085,176.848,20.670,153.053
C07916=1091.186,255.439,422.114,176.846,20.668,153.053
C07917=1091.180,255.191,422.140,176.843,20.666,153.053
C07918=1091.174,254.943,422.168,176.840,20.663,153.053
C07919=1091.169,254.694,422.195,176.836,20.661,153.053
C07920=1091.163,254.446,422.223,176.834,20.659,153.053
C07921=1091.157,254.197,422.250,176.831,20.656,153.053
C07922=1091.152,253.948,422.277,176.828,20.654,153.053
C07923=1091.146,253.701,422.305,176.824,20.651,153.053
C07924=1091.141,253.452,422.332,176.822,20.649,153.053
C07925=1091.136,253.203,422.359,176.819,20.647,153.053
C07926=1091.129,252.955,422.387,176.816,20.644,153.053
C07927=1091.124,252.706,422.414,176.813,20.642,153.053
C07928=1091.118,252.458,422.441,176.810,20.640,153.053
C07929=1091.113,252.209,422.468,176.807,20.637,153.053
C07930=1091.107,251.961,422.495,176.804,20.635,153.053
C07931=1091.102,251.713,422.523,176.801,20.633,153.053
C07932=1091.096,251.464,422.550,176.798,20.631,153.053
C07933=1091.090,251.215,422.576,176.795,20.628,153.053
C07934=1091.085,250.967,422.604,176.792,20.626,153.052
C07935=1091.079,250.719,422.631,176.790,20.624,153.052
C07936=1091.074,250.470,422.658,176.786,20.621,153.052
C07937=1091.068,250.222,422.685,176.783,20.619,153.052
C07938=1091.060,249.852,422.726,176.779,20.615,153.052
C07939=1091.052,249.483,422.765,176.774,20.612,153.052
C07940=1091.043,249.115,422.805,176.771,20.608,153.052
C07941=1091.035,248.746,422.845,176.766,20.604,153.052
C07942=1091.030,248.497,422.873,176.764,20.602,153.052
C07943=1091.024,248.249,422.899,176.760,20.600,153.052
C07944=1091.019,248.000,422.926,176.757,20.597,153.052
C07945=1091.013,247.752,422.953,176.754,20.595,153.052
C07946=1091.008,247.503,422.980,176.752,20.593,153.052
C07947=1091.002,247.254,423.007,176.748,20.590,153.052
C07948=1090.996,247.006,423.034,176.745,20.588,153.052
C07949=1090.990,246.758,423.061,176.743,20.586,153.052
C07950=1090.985,246.509,423.088,176.740,20.584,153.052
C07951=1090.980,246.261,423.115,176.736,20.582,153.052
C07952=1090.974,246.012,423.141,176.734,20.580,153.052
C07953=1090.968,245.763,423.167,176.731,20.577,153.052
C07954=1090.963,245.515,423.194,176.728,20.575,153.052
C07955=1090.958,245.266,423.221,176.725,20.573,153.052
C07956=1090.952,245.018,423.248,176.722,20.570,153.052
C07957=1090.946,244.770,423.274,176.719,20.568,153.052
C07958=1090.940,244.521,423.301,176.716,20.566,153.052
C07959=1090.935,244.273,423.328,176.713,20.563,153.052
C07960=1090.930,244.024,423.354,176.710,20.561,153.052
C07961=1090.924,243.775,423.381,176.708,20.559,153.052
C07962=1090.918,243.527,423.407,176.705,20.556,153.052
C07963=1090.912,243.278,423.434,176.701,20.554,153.052
C07964=1090.907,243.030,423.461,176.699,20.552,153.052
C07965=1090.902,242.781,423.487,176.696,20.549,153.052
C07966=1090.896,242.532,423.514,176.692,20.547,153.052
C07967=1090.890,242.284,423.541,176.690,20.545,153.052
C07968=1090.885,242.036,423.567,176.687,20.543,153.052
C07969=1090.879,241.787,423.593,176.684,20.540,153.052
C07970=1090.873,241.538,423.620,176.681,20.538,153.051
C07971=1090.868,241.290,423.646,176.678,20.536,153.051
C07972=1090.862,241.041,423.672,176.675,20.533,153.051
C07973=1090.856,240.793,423.699,176.672,20.532,153.052
C07974=1090.851,240.544,423.726,176.669,20.529,153.052
C07975=1090.845,240.295,423.752,176.666,20.527,153.052
C07976=1090.839,240.047,423.778,176.664,20.525,153.051
C07977=1090.834,239.798,423.804,176.660,20.522,153.051
C07978=1090.828,239.550,423.831,176.657,20.520,153.051
C07979=1090.822,239.301,423.857,176.655,20.518,153.051
C07980=1090.817,239.052,423.883,176.651,20.516,153.052
C07981=1090.811,238.804,423.910,176.649,20.514,153.051
C07982=1090.805,238.555,423.935,176.646,20.512,153.051
C07983=1090.799,238.307,423.962,176.643,20.509,153.051
C07984=1090.794,238.058,423.988,176.640,20.507,153.051
C07985=1090.788,237.810,424.014,176.637,20.505,153.051
C07986=1090.783,237.561,424.040,176.634,20.503,153.052
C07987=1090.777,237.313,424.067,176.631,20.501,153.051
C07988=1090.772,237.064,424.093,176.628,20.498,153.051
C07989=1090.766,236.816,424.119,176.626,20.496,153.051
C07990=1090.758,236.440,424.159,176.621,20.493,153.051
C07991=1090.749,236.064,424.198,176.617,20.489,153.051
C07992=1090.740,235.688,424.237,176.612,20.486,153.051
C07993=1090.732,235.312,424.276,176.608,20.483,153.051
C07994=1090.726,235.064,424.303,176.605,20.480,153.051
C07995=1090.721,234.815,424.329,176.602,20.478,153.051
C07996=1090.715,234.566,424.355,176.600,20.476,153.051
C07997=1090.710,234.317,424.381,176.596,20.473,153.051
C07998=1090.705,234.069,424.407,176.594,20.471,153.051
C07999=1090.699,233.820,424.432,176.591,20.469,153.051
C08000=1090.693,233.572,424.459,176.587,20.467,153.051
C08001=1090.687,233.323,424.485,176.585,20.465,153.051
C08002=1090.682,233.074,424.511,176.582,20.462,153.051
C08003=1090.676,232.826,424.536,176.580,20.460,153.051
C08004=1090.671,232.578,424.562,176.576,20.458,153.051
C08005=1090.665,232.329,424.588,176.573,20.456,153.051
C08006=1090.660,232.080,424.614,176.571,20.454,153.051
C08007=1090.653,231.831,424.640,176.567,20.451,153.051
C08008=1090.648,231.583,424.665,176.565,20.449,153.051
C08009=1090.643,231.334,424.691,176.562,20.447,153.051
C08010=1090.637,231.086,424.717,176.560,20.445,153.051
C08011=1090.631,230.837,424.743,176.556,20.443,153.051
C08012=1090.626,230.588,424.769,176.553,20.440,153.051
C08013=1090.620,230.340,424.794,176.551,20.439,153.051
C08014=1090.615,230.091,424.820,176.547,20.436,153.051
C08015=1090.609,229.842,424.846,176.545,20.434,153.051
C08016=1090.603,229.593,424.871,176.542,20.432,153.051
C08017=1090.598,229.345,424.897,176.538,20.430,153.051
C08018=1090.592,229.096,424.922,176.536,20.428,153.051
C08019=1090.586,228.847,424.948,176.533,20.425,153.051
C08020=1090.580,228.599,424.973,176.530,20.424,153.051
C08021=1090.575,228.350,424.999,176.527,20.421,153.051
C08022=1090.569,228.102,425.024,176.525,20.419,153.051
C08023=1090.564,227.853,425.050,176.522,20.417,153.051
C08024=1090.558,227.605,425.075,176.519,20.415,153.051
C08025=1090.552,227.356,425.101,176.516,20.413,153.051
C08026=1090.546,227.107,425.126,176.513,20.410,153.051
C08027=1090.541,226.858,425.152,176.510,20.408,153.051
C08028=1090.535,226.610,425.177,176.507,20.406,153.051
C08029=1090.530,226.361,425.203,176.505,20.404,153.051
C08030=1090.524,226.112,425.229,176.501,20.402,153.051
C08031=1090.519,225.864,425.254,176.499,20.400,153.051
C08032=1090.512,225.615,425.279,176.496,20.397,153.051
C08033=1090.507,225.366,425.305,176.494,20.395,153.051
C08034=1090.502,225.118,425.330,176.490,20.393,153.051
C08035=1090.496,224.869,425.356,176.487,20.391,153.051
C08036=1090.490,224.620,425.381,176.485,20.389,153.051
C08037=1090.485,224.372,425.406,176.481,20.386,153.051
C08038=1090.479,224.123,425.432,176.479,20.384,153.051
C08039=1090.474,223.874,425.457,176.476,20.382,153.051
C08040=1090.468,223.626,425.482,176.473,20.380,153.051
C08041=1090.463,223.377,425.508,176.470,20.378,153.051
C08042=1090.454,222.992,425.547,176.466,20.375,153.051
C08043=1090.445,222.608,425.586,176.461,20.371,153.051
C08044=1090.437,222.224,425.624,176.457,20.368,153.051
C08045=1090.428,221.839,425.663,176.453,20.364,153.051
C08046=1090.422,221.590,425.689,176.450,20.362,153.051
C08047=1090.417,221.342,425.713,176.447,20.360,153.052
C08048=1090.411,221.093,425.739,176.444,20.358,153.051
C08049=1090.405,220.845,425.764,176.441,20.356,153.051
C08050=1090.400,220.595,425.789,176.439,20.354,153.051
C08051=1090.394,220.347,425.814,176.436,20.352,153.052
C08052=1090.389,220.098,425.838,176.433,20.350,153.052
C08053=1090.382,219.850,425.864,176.430,20.347,153.052
C08054=1090.378,219.601,425.889,176.428,20.345,153.051
C08055=1090.372,219.352,425.914,176.424,20.343,153.052
C08056=1090.366,219.104,425.939,176.422,20.341,153.052
C08057=1090.360,218.855,425.964,176.419,20.339,153.052
C08058=1090.354,218.606,425.989,176.416,20.337,153.052
C08059=1090.349,218.357,426.014,176.413,20.335,153.052
C08060=1090.343,218.108,426.039,176.411,20.333,153.052
C08061=1090.338,217.860,426.063,176.408,20.330,153.052
C08062=1090.332,217.611,426.089,176.405,20.328,153.052
C08063=1090.326,217.363,426.113,176.402,20.326,153.052
C08064=1090.321,217.114,426.139,176.399,20.324,153.052
C08065=1090.316,216.865,426.163,176.396,20.322,153.052
C08066=1090.310,216.616,426.188,176.394,20.320,153.052
C08067=1090.304,216.368,426.213,176.391,20.318,153.052
C08068=1090.298,216.119,426.237,176.388,20.316,153.052
C08069=1090.293,215.871,426.262,176.385,20.314,153.052
C08070=1090.287,215.622,426.287,176.383,20.312,153.052
C08071=1090.282,215.372,426.312,176.379,20.310,153.052
C08072=1090.277,215.124,426.337,176.377,20.308,153.052
C08073=1090.271,214.875,426.361,176.374,20.305,153.052
C08074=1090.265,214.627,426.386,176.371,20.303,153.052
C08075=1090.259,214.378,426.411,176.368,20.301,153.052
C08076=1090.254,214.129,426.435,176.366,20.299,153.052
C08077=1090.249,213.881,426.459,176.362,20.297,153.052
C08078=1090.242,213.632,426.485,176.360,20.295,153.052
C08079=1090.237,213.383,426.509,176.358,20.293,153.052
C08080=1090.231,213.134,426.534,176.354,20.291,153.052
C08081=1090.226,212.886,426.558,176.352,20.289,153.052
C08082=1090.220,212.637,426.583,176.349,20.286,153.052
C08083=1090.214,212.388,426.608,176.347,20.284,153.052
C08084=1090.209,212.140,426.632,176.343,20.282,153.052
C08085=1090.203,211.890,426.656,176.341,20.280,153.052
C08086=1090.198,211.642,426.681,176.338,20.278,153.052
C08087=1090.192,211.393,426.705,176.335,20.276,153.052
C08088=1090.186,211.145,426.730,176.332,20.274,153.052
C08089=1090.181,210.896,426.754,176.330,20.272,153.052
C08090=1090.175,210.647,426.779,176.326,20.269,153.052
C08091=1090.170,210.398,426.803,176.324,20.267,153.052
C08092=1090.165,210.150,426.828,176.322,20.266,153.052
C08093=1090.159,209.900,426.852,176.318,20.263,153.052
C08094=1090.150,209.520,426.890,176.314,20.260,153.052
C08095=1090.142,209.139,426.927,176.310,20.257,153.052
C08096=1090.133,208.759,426.964,176.305,20.254,153.052
C08097=1090.124,208.378,427.001,176.302,20.250,153.052
C08098=1090.101,207.356,427.100,176.233,20.217,153.056
C08099=1090.096,207.107,427.124,176.231,20.216,153.056
C08100=1090.090,206.859,427.147,176.228,20.215,153.057
C08101=1090.085,206.610,427.171,176.225,20.213,153.057
C08102=1090.079,206.361,427.196,176.222,20.212,153.057
C08103=1090.073,206.112,427.219,176.219,20.211,153.057
C08104=1090.068,205.863,427.243,176.216,20.210,153.058
C08105=1090.062,205.615,427.266,176.213,20.209,153.058
C08106=1090.057,205.366,427.291,176.211,20.208,153.058
C08107=1090.052,205.117,427.314,176.208,20.206,153.058
C08108=1090.045,204.868,427.338,176.204,20.205,153.058
C08109=1090.040,204.619,427.363,176.202,20.204,153.059
C08110=1090.034,204.371,427.385,176.199,20.203,153.059
C08111=1090.029,204.122,427.410,176.196,20.202,153.059
C08112=1090.024,203.873,427.433,176.193,20.200,153.059
C08113=1090.018,203.624,427.457,176.191,20.199,153.060
C08114=1090.012,203.376,427.481,176.187,20.198,153.060
C08115=1090.006,203.126,427.504,176.184,20.197,153.060
C08116=1090.001,202.878,427.529,176.182,20.195,153.060
C08117=1089.995,202.629,427.552,176.179,20.194,153.060
C08118=1089.990,202.380,427.576,176.176,20.193,153.061
C08119=1089.984,202.131,427.599,176.173,20.192,153.061
C08120=1089.979,201.883,427.623,176.171,20.191,153.061
C08121=1089.973,201.634,427.646,176.167,20.189,153.062
C08122=1089.966,201.385,427.670,176.164,20.188,153.062
C08123=1089.961,201.136,427.694,176.161,20.187,153.062
C08124=1089.955,200.887,427.717,176.159,20.186,153.062
C08125=1089.950,200.638,427.740,176.156,20.185,153.062
C08126=1089.945,200.389,427.764,176.153,20.184,153.063
C08127=1089.939,200.141,427.787,176.150,20.183,153.063
C08128=1089.934,199.892,427.811,176.147,20.181,153.063
C08129=1089.928,199.643,427.835,176.144,20.180,153.063
C08130=1089.921,199.394,427.858,176.141,20.179,153.064
C08131=1089.916,199.145,427.882,176.139,20.178,153.064
C08132=1089.910,198.896,427.905,176.136,20.177,153.064
C08133=1089.904,198.647,427.928,176.133,20.176,153.064
C08134=1089.899,198.398,427.952,176.130,20.175,153.065
C08135=1089.893,198.150,427.975,176.128,20.174,153.065
C08136=1089.888,197.901,427.998,176.124,20.172,153.065
C08137=1089.882,197.652,428.021,176.121,20.171,153.065
C08138=1089.877,197.404,428.045,176.119,20.170,153.065
C08139=1089.871,197.155,428.068,176.116,20.169,153.066
C08140=1089.865,196.906,428.091,176.113,20.168,153.066
C08141=1089.860,196.657,428.116,176.110,20.166,153.066
C08142=1089.854,196.408,428.139,176.108,20.165,153.066
C08143=1089.848,196.159,428.162,176.105,20.164,153.067
C08144=1089.843,195.911,428.184,176.102,20.163,153.067
C08145=1089.838,195.661,428.208,176.099,20.162,153.067
C08146=1089.832,195.413,428.232,176.096,20.160,153.067
C08147=1089.826,195.164,428.255,176.093,20.159,153.067
C08148=1089.821,194.915,428.278,176.090,20.158,153.068
C08149=1089.815,194.666,428.301,176.088,20.157,153.068
C08150=1089.809,194.417,428.324,176.085,20.156,153.068
C08151=1089.804,194.168,428.347,176.082,20.155,153.068
C08152=1089.798,193.920,428.371,176.079,20.154,153.069
C08153=1089.793,193.671,428.394,176.077,20.152,153.069
C08154=1089.787,193.422,428.417,176.074,20.151,153.069
C08155=1089.781,193.173,428.440,176.071,20.150,153.069
C08156=1089.776,192.924,428.463,176.068,20.149,153.069
C08157=1089.771,192.675,428.487,176.065,20.147,153.070
C08158=1089.765,192.426,428.510,176.062,20.146,153.070
C08159=1089.758,192.150,428.535,176.060,20.145,153.070
C08160=1089.752,191.873,428.561,176.057,20.144,153.070
C08161=1089.746,191.596,428.586,176.053,20.142,153.070
C08162=1089.740,191.319,428.612,176.051,20.141,153.071
C08163=1089.734,191.070,428.635,176.048,20.140,153.071
C08164=1089.729,190.821,428.658,176.045,20.138,153.071
C08165=1089.724,190.572,428.681,176.042,20.137,153.071
C08166=1089.718,190.323,428.704,176.039,20.136,153.072
C08167=1089.712,190.074,428.727,176.036,20.134,153.072
C08168=1089.707,189.825,428.750,176.033,20.133,153.072
C08169=1089.702,189.577,428.773,176.031,20.132,153.072
C08170=1089.696,189.328,428.796,176.028,20.131,153.072
C08171=1089.691,189.079,428.819,176.025,20.130,153.073
C08172=1089.685,188.830,428.842,176.023,20.128,153.073
C08173=1089.679,188.581,428.865,176.020,20.127,153.073
C08174=1089.673,188.332,428.888,176.017,20.126,153.073
C08175=1089.669,188.084,428.910,176.015,20.125,153.073
C08176=1089.664,187.834,428.933,176.012,20.124,153.074
C08177=1089.658,187.585,428.956,176.009,20.122,153.074
C08178=1089.652,187.337,428.979,176.006,20.121,153.074
C08179=1089.646,187.088,429.002,176.004,20.120,153.074
C08180=1089.641,186.840,429.025,176.001,20.119,153.074
C08181=1089.636,186.590,429.047,175.998,20.118,153.075
C08182=1089.630,186.341,429.070,175.996,20.116,153.075
C08183=1089.624,186.092,429.093,175.993,20.115,153.075
C08184=1089.619,185.843,429.116,175.990,20.114,153.075
C08185=1089.614,185.595,429.138,175.988,20.113,153.075
C08186=1089.609,185.345,429.161,175.984,20.111,153.076
C08187=1089.603,185.096,429.184,175.981,20.110,153.076
C08188=1089.597,184.848,429.206,175.979,20.109,153.076
C08189=1089.591,184.599,429.229,175.976,20.108,153.076
C08190=1089.586,184.350,429.251,175.973,20.106,153.076
C08191=1089.580,184.101,429.274,175.971,20.105,153.077
C08192=1089.574,183.853,429.296,175.968,20.104,153.077
C08193=1089.569,183.603,429.319,175.965,20.103,153.077
C08194=1089.563,183.354,429.342,175.962,20.102,153.077
C08195=1089.557,183.105,429.365,175.960,20.101,153.077
C08196=1089.551,182.856,429.386,175.957,20.100,153.078
C08197=1089.546,182.608,429.409,175.954,20.099,153.078
C08198=1089.540,182.359,429.432,175.952,20.097,153.078
C08199=1089.535,182.109,429.454,175.949,20.096,153.078
C08200=1089.528,181.861,429.476,175.946,20.095,153.079
C08201=1089.523,181.611,429.499,175.943,20.094,153.079
C08202=1089.518,181.363,429.521,175.941,20.093,153.079
C08203=1089.512,181.114,429.544,175.938,20.092,153.079
C08204=1089.506,180.865,429.566,175.935,20.090,153.079
C08205=1089.500,180.616,429.589,175.933,20.089,153.080
C08206=1089.495,180.367,429.611,175.930,20.088,153.080
C08207=1089.489,180.119,429.633,175.927,20.086,153.080
C08208=1089.483,179.869,429.655,175.924,20.085,153.080
C08209=1089.478,179.620,429.678,175.922,20.084,153.081
C08210=1089.471,179.371,429.700,175.919,20.083,153.081
C08211=1089.466,179.123,429.722,175.916,20.082,153.081
C08212=1089.461,178.873,429.744,175.913,20.081,153.081
C08213=1089.454,178.625,429.767,175.911,20.079,153.081
C08214=1089.449,178.375,429.789,175.908,20.078,153.082
C08215=1089.444,178.127,429.812,175.906,20.077,153.082
C08216=1089.438,177.878,429.833,175.903,20.076,153.082
C08217=1089.432,177.628,429.855,175.900,20.075,153.082
C08218=1089.426,177.380,429.878,175.897,20.073,153.082
C08219=1089.421,177.131,429.900,175.896,20.073,153.082
C08220=1089.415,176.882,429.923,175.893,20.071,153.083
C08221=1089.410,176.633,429.945,175.890,20.070,153.083
C08222=1089.404,176.384,429.966,175.887,20.069,153.083
C08223=1089.398,176.107,429.991,175.884,20.067,153.083
C08224=1089.391,175.830,430.016,175.881,20.066,153.084
C08225=1089.385,175.552,430.041,175.879,20.065,153.084
C08226=1089.378,175.275,430.065,175.875,20.063,153.084
C08227=1089.374,175.026,430.087,175.872,20.062,153.084
C08228=1089.368,174.778,430.110,175.870,20.061,153.084
C08229=1089.362,174.528,430.132,175.867,20.060,153.085
C08230=1089.357,174.280,430.154,175.865,20.059,153.085
C08231=1089.351,174.030,430.175,175.862,20.058,153.085
C08232=1089.346,173.782,430.198,175.860,20.056,153.085
C08233=1089.340,173.533,430.220,175.857,20.055,153.085
C08234=1089.334,173.283,430.242,175.854,20.054,153.085
C08235=1089.329,173.035,430.263,175.852,20.053,153.086
C08236=1089.323,172.786,430.286,175.849,20.051,153.086
C08237=1089.318,172.537,430.308,175.846,20.050,153.086
C08238=1089.312,172.288,430.329,175.844,20.049,153.086
C08239=1089.306,172.038,430.352,175.841,20.048,153.086
C08240=1089.301,171.790,430.373,175.838,20.046,153.086
C08241=1089.295,171.540,430.395,175.836,20.045,153.087
C08242=1089.290,171.292,430.418,175.833,20.044,153.087
C08243=1089.284,171.043,430.439,175.831,20.042,153.087
C08244=1089.279,170.794,430.461,175.828,20.041,153.087
C08245=1089.273,170.545,430.483,175.825,20.040,153.087
C08246=1089.268,170.295,430.505,175.822,20.039,153.088
C08247=1089.262,170.047,430.526,175.820,20.037,153.088
C08248=1089.257,169.797,430.549,175.818,20.036,153.088
C08249=1089.251,169.549,430.570,175.815,20.035,153.088
C08250=1089.246,169.299,430.592,175.813,20.034,153.088
C08251=1089.240,169.051,430.613,175.810,20.033,153.088
C08252=1089.234,168.802,430.636,175.807,20.031,153.089
C08253=1089.229,168.554,430.657,175.805,20.030,153.089
C08254=1089.223,168.304,430.680,175.802,20.029,153.089
C08255=1089.218,168.056,430.701,175.800,20.027,153.089
C08256=1089.212,167.806,430.723,175.797,20.026,153.089
C08257=1089.207,167.558,430.744,175.794,20.025,153.089
C08258=1089.201,167.308,430.767,175.792,20.023,153.090
C08259=1089.196,167.059,430.788,175.789,20.022,153.090
C08260=1089.190,166.810,430.810,175.786,20.021,153.090
C08261=1089.185,166.561,430.831,175.784,20.019,153.090
C08262=1089.180,166.312,430.853,175.782,20.018,153.090
C08263=1089.174,166.063,430.874,175.779,20.017,153.090
C08264=1089.169,165.814,430.896,175.777,20.016,153.091
C08265=1089.163,165.565,430.918,175.774,20.014,153.091
C08266=1089.158,165.316,430.939,175.771,20.013,153.091
C08267=1089.152,165.067,430.961,175.769,20.012,153.091
C08268=1089.147,164.818,430.983,175.766,20.010,153.091
C08269=1089.142,164.569,431.004,175.764,20.009,153.091
C08270=1089.136,164.320,431.026,175.761,20.008,153.092
C08271=1089.131,164.071,431.047,175.758,20.006,153.092
C08272=1089.125,163.822,431.069,175.757,20.005,153.092
C08273=1089.119,163.573,431.090,175.754,20.004,153.092
C08274=1089.115,163.324,431.112,175.751,20.003,153.092
C08275=1089.108,163.075,431.134,175.749,20.001,153.092
C08276=1089.104,162.826,431.155,175.746,20.000,153.092
C08277=1089.098,162.577,431.176,175.744,19.998,153.092
C08278=1089.092,162.328,431.198,175.741,19.997,153.093
C08279=1089.087,162.079,431.220,175.738,19.996,153.093
C08280=1089.081,161.829,431.240,175.736,19.994,153.093
C08281=1089.077,161.580,431.262,175.733,19.993,153.093
C08282=1089.071,161.332,431.284,175.731,19.992,153.093
C08283=1089.065,161.083,431.305,175.729,19.991,153.093
C08284=1089.060,160.834,431.326,175.726,19.989,153.094
C08285=1089.054,160.584,431.347,175.723,19.988,153.094
C08286=1089.048,160.336,431.369,175.721,19.987,153.094
C08287=1089.042,160.056,431.392,175.718,19.985,153.094
C08288=1089.036,159.777,431.416,175.716,19.984,153.094
C08289=1089.029,159.496,431.440,175.712,19.982,153.094
C08290=1089.023,159.217,431.464,175.710,19.981,153.095
C08291=1089.017,158.968,431.486,175.707,19.980,153.095
C08292=1089.012,158.719,431.506,175.704,19.978,153.095
C08293=1089.006,158.470,431.528,175.703,19.977,153.095
C08294=1089.001,158.221,431.549,175.700,19.976,153.095
C08295=1088.995,157.972,431.570,175.697,19.975,153.095
C08296=1088.989,157.723,431.592,175.695,19.973,153.096
C08297=1088.984,157.474,431.612,175.692,19.972,153.096
C08298=1088.978,157.225,431.633,175.689,19.971,153.096
C08299=1088.973,156.975,431.655,175.687,19.969,153.096
C08300=1088.967,156.727,431.676,175.685,19.968,153.096
C08301=1088.962,156.477,431.697,175.682,19.967,153.096
C08302=1088.956,156.228,431.718,175.680,19.965,153.096
C08303=1088.951,155.979,431.739,175.677,19.964,153.097
C08304=1088.945,155.731,431.760,175.675,19.963,153.097
C08305=1088.939,155.481,431.781,175.672,19.961,153.097
C08306=1088.934,155.232,431.802,175.669,19.960,153.097
C08307=1088.928,154.983,431.823,175.668,19.959,153.097
C08308=1088.922,154.734,431.845,175.665,19.958,153.097
C08309=1088.917,154.485,431.865,175.662,19.956,153.097
C08310=1088.911,154.236,431.886,175.660,19.955,153.098
C08311=1088.906,153.987,431.907,175.657,19.954,153.098
C08312=1088.900,153.738,431.929,175.655,19.952,153.098
C08313=1088.895,153.489,431.949,175.653,19.951,153.098
C08314=1088.890,153.240,431.970,175.650,19.950,153.098
C08315=1088.883,152.991,431.991,175.648,19.948,153.098
C08316=1088.877,152.742,432.011,175.645,19.947,153.099
C08317=1088.872,152.493,432.033,175.642,19.946,153.099
C08318=1088.866,152.243,432.053,175.640,19.944,153.099
C08319=1088.861,151.994,432.074,175.638,19.943,153.099
C08320=1088.855,151.746,432.095,175.636,19.942,153.099
C08321=1088.850,151.497,432.116,175.633,19.940,153.099
C08322=1088.844,151.247,432.137,175.630,19.939,153.099
C08323=1088.838,150.998,432.158,175.628,19.938,153.099
C08324=1088.833,150.749,432.179,175.625,19.936,153.100
C08325=1088.828,150.500,432.199,175.623,19.935,153.100
C08326=1088.822,150.251,432.221,175.621,19.934,153.100
C08327=1088.816,150.002,432.241,175.618,19.932,153.100
C08328=1088.811,149.753,432.261,175.616,19.931,153.100
C08329=1088.805,149.504,432.282,175.613,19.929,153.100
C08330=1088.800,149.255,432.303,175.610,19.928,153.100
C08331=1088.794,149.005,432.324,175.609,19.927,153.101
C08332=1088.789,148.756,432.345,175.606,19.926,153.101
C08333=1088.783,148.507,432.365,175.604,19.924,153.101
C08334=1088.777,148.258,432.385,175.601,19.923,153.101
C08335=1088.772,148.010,432.406,175.598,19.921,153.101
C08336=1088.766,147.762,432.427,175.597,19.920,153.101
C08337=1088.760,147.514,432.447,175.594,19.919,153.101
C08338=1088.755,147.267,432.468,175.591,19.918,153.101
C08339=1088.749,147.018,432.488,175.589,19.916,153.102
C08340=1088.743,146.770,432.509,175.586,19.915,153.102
C08341=1088.738,146.522,432.529,175.585,19.914,153.102
C08342=1088.732,146.274,432.550,175.582,19.912,153.102
C08343=1088.727,146.025,432.571,175.580,19.911,153.102
C08344=1088.721,145.776,432.591,175.577,19.909,153.102
C08345=1088.715,145.527,432.611,175.574,19.908,153.102
C08346=1088.710,145.278,432.632,175.573,19.907,153.102
C08347=1088.705,145.029,432.652,175.570,19.905,153.103
C08348=1088.698,144.779,432.673,175.567,19.904,153.103
C08349=1088.693,144.530,432.693,175.565,19.903,153.103
C08350=1088.688,144.281,432.714,175.563,19.902,153.103
C08351=1088.681,144.004,432.736,175.560,19.900,153.103
C08352=1088.675,143.726,432.759,175.557,19.898,153.103
C08353=1088.669,143.448,432.782,175.555,19.897,153.103
C08354=1088.662,143.171,432.805,175.552,19.895,153.104
C08355=1088.657,142.921,432.825,175.549,19.894,153.104
C08356=1088.652,142.672,432.846,175.548,19.893,153.104
C08357=1088.646,142.424,432.866,175.545,19.891,153.104
C08358=1088.640,142.174,432.887,175.543,19.890,153.104
C08359=1088.635,141.925,432.907,175.540,19.888,153.104
C08360=1088.629,141.676,432.927,175.538,19.887,153.104
C08361=1088.624,141.427,432.948,175.536,19.886,153.104
C08362=1088.618,141.178,432.968,175.533,19.884,153.104
C08363=1088.613,140.928,432.988,175.531,19.883,153.105
C08364=1088.607,140.679,433.008,175.528,19.881,153.105
C08365=1088.601,140.430,433.028,175.526,19.880,153.105
C08366=1088.596,140.181,433.049,175.524,19.879,153.105
C08367=1088.590,139.932,433.069,175.521,19.877,153.105
C08368=1088.585,139.683,433.089,175.519,19.876,153.105
C08369=1088.579,139.434,433.109,175.516,19.874,153.105
C08370=1088.573,139.184,433.130,175.515,19.873,153.105
C08371=1088.567,138.935,433.149,175.512,19.872,153.105
C08372=1088.562,138.686,433.170,175.509,19.870,153.106
C08373=1088.556,138.437,433.190,175.507,19.868,153.106
C08374=1088.551,138.188,433.210,175.505,19.867,153.106
C08375=1088.545,137.939,433.230,175.503,19.866,153.106
C08376=1088.540,137.689,433.250,175.500,19.864,153.106
C08377=1088.534,137.441,433.270,175.498,19.863,153.106
C08378=1088.529,137.191,433.291,175.496,19.862,153.106
C08379=1088.523,136.943,433.311,175.494,19.860,153.106
C08380=1088.517,136.694,433.331,175.491,19.859,153.106
C08381=1088.512,136.444,433.350,175.488,19.857,153.107
C08382=1088.506,136.195,433.370,175.487,19.856,153.107
C08383=1088.500,135.946,433.391,175.484,19.855,153.107
C08384=1088.495,135.697,433.410,175.482,19.853,153.107
C08385=1088.489,135.448,433.431,175.479,19.852,153.107
C08386=1088.483,135.199,433.451,175.477,19.851,153.107
C08387=1088.477,134.950,433.471,175.475,19.849,153.107
C08388=1088.473,134.700,433.490,175.472,19.847,153.107
C08389=1088.467,134.451,433.510,175.470,19.846,153.107
C08390=1088.461,134.202,433.531,175.468,19.845,153.107
C08391=1088.456,133.953,433.550,175.466,19.843,153.107
C08392=1088.450,133.704,433.570,175.463,19.842,153.108
C08393=1088.445,133.454,433.590,175.461,19.840,153.108
C08394=1088.439,133.206,433.610,175.459,19.839,153.108
C08395=1088.433,132.956,433.630,175.457,19.837,153.108
C08396=1088.428,132.707,433.650,175.454,19.836,153.108
C08397=1088.422,132.458,433.670,175.452,19.835,153.108
C08398=1088.417,132.208,433.690,175.450,19.833,153.108
C08399=1088.411,131.960,433.709,175.447,19.832,153.108
C08400=1088.405,131.711,433.729,175.445,19.830,153.108
C08401=1088.399,131.461,433.749,175.443,19.829,153.108
C08402=1088.393,131.213,433.769,175.440,19.828,153.109
C08403=1088.388,130.963,433.788,175.438,19.826,153.109
C08404=1088.382,130.714,433.808,175.436,19.824,153.109
C08405=1088.376,130.465,433.828,175.434,19.823,153.109
C08406=1088.370,130.216,433.848,175.431,19.822,153.109
C08407=1088.365,129.966,433.867,175.429,19.820,153.109
C08408=1088.359,129.717,433.887,175.427,19.819,153.109
C08409=1088.354,129.468,433.907,175.424,19.818,153.109
C08410=1088.348,129.219,433.927,175.422,19.816,153.109
C08411=1088.342,128.969,433.946,175.420,19.814,153.109
C08412=1088.336,128.721,433.966,175.418,19.813,153.109
C08413=1088.330,128.471,433.985,175.415,19.812,153.110
C08414=1088.325,128.222,434.004,175.413,19.810,153.110
C08415=1088.319,127.945,434.026,175.410,19.809,153.110
C08416=1088.312,127.667,434.048,175.408,19.807,153.110
C08417=1088.306,127.389,434.070,175.405,19.805,153.110
C08418=1088.299,127.111,434.092,175.403,19.804,153.110
C08419=1088.294,126.862,434.112,175.401,19.803,153.110
C08420=1088.289,126.612,434.131,175.399,19.801,153.110
C08421=1088.283,126.363,434.151,175.396,19.799,153.110
C08422=1088.277,126.114,434.171,175.394,19.798,153.110
C08423=1088.272,125.865,434.189,175.392,19.797,153.111
C08424=1088.266,125.616,434.209,175.389,19.795,153.111
C08425=1088.260,125.367,434.229,175.387,19.794,153.111
C08426=1088.254,125.117,434.248,175.385,19.792,153.111
C08427=1088.249,124.868,434.267,175.383,19.791,153.111
C08428=1088.243,124.619,434.286,175.380,19.789,153.111
C08429=1088.238,124.369,434.307,175.379,19.788,153.111
C08430=1088.233,124.121,434.326,175.376,19.786,153.111
C08431=1088.227,123.871,434.345,175.374,19.785,153.111
C08432=1088.221,123.623,434.365,175.371,19.783,153.111
C08433=1088.215,123.373,434.384,175.370,19.782,153.111
C08434=1088.210,123.124,434.403,175.367,19.780,153.111
C08435=1088.204,122.874,434.423,175.365,19.779,153.112
C08436=1088.199,122.625,434.442,175.363,19.777,153.111
C08437=1088.193,122.377,434.462,175.361,19.776,153.112
C08438=1088.187,122.127,434.481,175.358,19.774,153.112
C08439=1088.181,121.878,434.500,175.357,19.773,153.112
C08440=1088.176,121.628,434.519,175.354,19.771,153.112
C08441=1088.171,121.380,434.538,175.351,19.770,153.112
C08442=1088.165,121.131,434.558,175.350,19.768,153.112
C08443=1088.159,120.881,434.577,175.347,19.767,153.112
C08444=1088.153,120.632,434.597,175.345,19.765,153.112
C08445=1088.148,120.383,434.616,175.343,19.764,153.112
C08446=1088.143,120.134,434.635,175.341,19.762,153.112
C08447=1088.137,119.884,434.654,175.339,19.760,153.112
C08448=1088.131,119.635,434.673,175.337,19.759,153.112
C08449=1088.125,119.385,434.692,175.334,19.758,153.112
C08450=1088.120,119.137,434.711,175.332,19.756,153.112
C08451=1088.115,118.887,434.731,175.330,19.755,153.112
C08452=1088.109,118.639,434.751,175.328,19.753,153.112
C08453=1088.104,118.390,434.769,175.325,19.751,153.113
C08454=1088.098,118.140,434.789,175.324,19.750,153.113
C08455=1088.092,117.891,434.808,175.321,19.748,153.113
C08456=1088.087,117.641,434.827,175.319,19.747,153.113
C08457=1088.081,117.393,434.846,175.317,19.745,153.113
C08458=1088.076,117.143,434.865,175.315,19.744,153.113
C08459=1088.070,116.894,434.885,175.313,19.742,153.113
C08460=1088.065,116.645,434.903,175.311,19.741,153.113
C08461=1088.059,116.396,434.923,175.308,19.739,153.113
C08462=1088.054,116.146,434.942,175.306,19.737,153.113
C08463=1088.049,115.898,434.961,175.304,19.736,153.113
C08464=1088.043,115.648,434.980,175.302,19.734,153.113
C08465=1088.037,115.398,434.999,175.300,19.732,153.113
C08466=1088.032,115.149,435.017,175.298,19.731,153.113
C08467=1088.026,114.900,435.036,175.296,19.729,153.113
C08468=1088.020,114.651,435.055,175.293,19.728,153.113
C08469=1088.015,114.402,435.074,175.292,19.726,153.113
C08470=1088.010,114.153,435.093,175.289,19.725,153.113
C08471=1088.004,113.903,435.113,175.287,19.723,153.113
C08472=1087.999,113.654,435.132,175.285,19.722,153.113
C08473=1087.992,113.405,435.150,175.283,19.720,153.113
C08474=1087.987,113.155,435.169,175.280,19.718,153.114
C08475=1087.981,112.906,435.188,175.279,19.717,153.114
C08476=1087.976,112.657,435.207,175.276,19.715,153.114
C08477=1087.970,112.408,435.225,175.274,19.713,153.114
C08478=1087.964,112.159,435.245,175.272,19.712,153.114
C08479=1087.958,111.880,435.265,175.270,19.710,153.114
C08480=1087.952,111.603,435.286,175.267,19.709,153.114
C08481=1087.946,111.325,435.307,175.265,19.707,153.114
C08482=1087.939,111.047,435.328,175.262,19.705,153.114
C08483=1087.934,110.798,435.347,175.260,19.703,153.114
C08484=1087.928,110.549,435.366,175.258,19.702,153.114
C08485=1087.922,110.299,435.384,175.256,19.700,153.114
C08486=1087.917,110.050,435.403,175.254,19.699,153.114
C08487=1087.910,109.801,435.422,175.252,19.697,153.114
C08488=1087.905,109.552,435.441,175.249,19.696,153.114
C08489=1087.900,109.302,435.459,175.248,19.694,153.114
C08490=1087.893,109.053,435.478,175.245,19.693,153.114
C08491=1087.888,108.804,435.497,175.243,19.691,153.114
C08492=1087.883,108.554,435.515,175.241,19.690,153.114
C08493=1087.877,108.305,435.534,175.239,19.688,153.114
C08494=1087.871,108.057,435.553,175.237,19.686,153.115
C08495=1087.865,107.807,435.571,175.235,19.685,153.114
C08496=1087.860,107.557,435.590,175.233,19.683,153.114
C08497=1087.854,107.309,435.608,175.231,19.682,153.115
C08498=1087.848,107.059,435.627,175.229,19.680,153.115
C08499=1087.843,106.810,435.646,175.226,19.678,153.115
C08500=1087.837,106.561,435.664,175.225,19.677,153.115
C08501=1087.832,106.311,435.683,175.222,19.675,153.115
C08502=1087.826,106.063,435.701,175.221,19.674,153.115
C08503=1087.820,105.813,435.720,175.218,19.672,153.115
C08504=1087.815,105.564,435.738,175.216,19.670,153.115
C08505=1087.809,105.314,435.756,175.214,19.669,153.115
C08506=1087.804,105.065,435.775,175.212,19.667,153.115
C08507=1087.798,104.816,435.794,175.210,19.665,153.115
C08508=1087.793,104.567,435.812,175.208,19.664,153.115
C08509=1087.786,104.318,435.831,175.206,19.662,153.115
C08510=1087.781,104.068,435.849,175.204,19.661,153.115
C08511=1087.775,103.819,435.868,175.202,19.659,153.115
C08512=1087.770,103.569,435.886,175.199,19.657,153.115
C08513=1087.764,103.321,435.904,175.198,19.656,153.115
C08514=1087.759,103.071,435.923,175.195,19.654,153.115
C08515=1087.753,102.822,435.941,175.194,19.653,153.115
C08516=1087.747,102.572,435.960,175.191,19.651,153.115
C08517=1087.742,102.324,435.978,175.189,19.649,153.115
C08518=1087.736,102.074,435.997,175.187,19.648,153.115
C08519=1087.731,101.825,436.014,175.185,19.646,153.115
C08520=1087.725,101.575,436.033,175.184,19.644,153.115
C08521=1087.720,101.326,436.051,175.181,19.643,153.115
C08522=1087.714,101.077,436.070,175.179,19.641,153.115
C08523=1087.708,100.828,436.088,175.177,19.639,153.115
C08524=1087.702,100.579,436.106,175.175,19.638,153.115
C08525=1087.697,100.329,436.125,175.173,19.636,153.115
C08526=1087.691,100.080,436.143,175.171,19.634,153.115
C08527=1087.685,99.831,436.161,175.168,19.633,153.115
C08528=1087.680,99.581,436.179,175.167,19.631,153.115
C08529=1087.674,99.332,436.197,175.165,19.629,153.115
C08530=1087.668,99.083,436.216,175.163,19.628,153.115
C08531=1087.663,98.834,436.234,175.161,19.626,153.115
C08532=1087.657,98.584,436.252,175.159,19.625,153.115
C08533=1087.651,98.336,436.270,175.157,19.623,153.115
C08534=1087.646,98.085,436.288,175.154,19.621,153.115
C08535=1087.640,97.836,436.306,175.153,19.620,153.115
C08536=1087.634,97.587,436.325,175.150,19.618,153.116
C08537=1087.629,97.338,436.343,175.149,19.617,153.115
C08538=1087.623,97.088,436.361,175.147,19.615,153.115
C08539=1087.617,96.840,436.379,175.144,19.613,153.115
C08540=1087.612,96.591,436.397,175.143,19.612,153.116
C08541=1087.606,96.341,436.415,175.140,19.610,153.116
C08542=1087.601,96.092,436.433,175.139,19.608,153.115
C08543=1087.594,95.814,436.453,175.136,19.606,153.115
C08544=1087.588,95.536,436.473,175.134,19.604,153.115
C08545=1087.581,95.258,436.493,175.132,19.603,153.116
C08546=1087.575,94.980,436.513,175.129,19.601,153.116
C08547=1087.570,94.731,436.531,175.128,19.599,153.116
C08548=1087.564,94.481,436.549,175.126,19.597,153.116
C08549=1087.558,94.233,436.568,175.124,19.596,153.115
C08550=1087.552,93.983,436.586,175.122,19.594,153.116
C08551=1087.547,93.734,436.603,175.119,19.592,153.116
C08552=1087.542,93.484,436.621,175.118,19.591,153.116
C08553=1087.536,93.235,436.639,175.115,19.589,153.116
C08554=1087.530,92.986,436.657,175.114,19.587,153.115
C08555=1087.525,92.737,436.674,175.112,19.585,153.115
C08556=1087.519,92.487,436.694,175.110,19.584,153.116
C08557=1087.514,92.238,436.711,175.108,19.582,153.116
C08558=1087.508,91.989,436.729,175.105,19.580,153.116
C08559=1087.502,91.739,436.747,175.104,19.578,153.116
C08560=1087.496,91.490,436.764,175.102,19.576,153.116
C08561=1087.492,91.241,436.782,175.100,19.575,153.115
C08562=1087.486,90.991,436.800,175.098,19.573,153.116
C08563=1087.480,90.742,436.818,175.096,19.572,153.116
C08564=1087.474,90.492,436.836,175.094,19.570,153.116
C08565=1087.468,90.243,436.853,175.092,19.568,153.115
C08566=1087.463,89.994,436.871,175.090,19.566,153.115
C08567=1087.457,89.745,436.889,175.087,19.565,153.116
C08568=1087.451,89.496,436.906,175.086,19.563,153.116
C08569=1087.445,89.246,436.924,175.084,19.561,153.116
C08570=1087.440,88.997,436.942,175.082,19.560,153.115
C08571=1087.434,88.748,436.960,175.080,19.558,153.115
C08572=1087.428,88.498,436.977,175.078,19.557,153.116
C08573=1087.422,88.249,436.995,175.076,19.555,153.116
C08574=1087.417,88.000,437.013,175.074,19.553,153.116
C08575=1087.411,87.750,437.031,175.072,19.551,153.116
C08576=1087.405,87.501,437.048,175.071,19.550,153.115
C08577=1087.400,87.252,437.066,175.068,19.548,153.115
C08578=1087.394,87.002,437.084,175.066,19.546,153.115
C08579=1087.388,86.753,437.101,175.064,19.545,153.116
C08580=1087.383,86.504,437.119,175.062,19.543,153.116
C08581=1087.376,86.255,437.137,175.061,19.541,153.115
C08582=1087.371,86.005,437.154,175.058,19.539,153.115
C08583=1087.366,85.756,437.171,175.057,19.538,153.115
C08584=1087.360,85.507,437.189,175.055,19.536,153.115
C08585=1087.354,85.257,437.207,175.053,19.534,153.115
C08586=1087.349,85.008,437.224,175.051,19.532,153.115
C08587=1087.343,84.759,437.242,175.049,19.531,153.115
C08588=1087.337,84.509,437.260,175.047,19.529,153.115
C08589=1087.332,84.260,437.277,175.045,19.528,153.115
C08590=1087.326,84.011,437.294,175.043,19.526,153.115
C08591=1087.321,83.762,437.312,175.041,19.524,153.115
C08592=1087.315,83.512,437.330,175.039,19.522,153.115
C08593=1087.309,83.263,437.347,175.037,19.520,153.115
C08594=1087.303,83.013,437.363,175.035,19.519,153.115
C08595=1087.298,82.764,437.381,175.033,19.517,153.115
C08596=1087.291,82.515,437.399,175.032,19.515,153.115
C08597=1087.286,82.266,437.416,175.029,19.513,153.115
C08598=1087.281,82.016,437.433,175.028,19.512,153.115
C08599=1087.275,81.767,437.451,175.026,19.510,153.115
C08600=1087.270,81.518,437.468,175.024,19.508,153.115
C08601=1087.264,81.268,437.486,175.022,19.506,153.115
C08602=1087.258,81.018,437.503,175.020,19.505,153.115
C08603=1087.253,80.769,437.521,175.018,19.503,153.115
C08604=1087.247,80.520,437.538,175.017,19.501,153.115
C08605=1087.242,80.271,437.555,175.014,19.499,153.115
C08606=1087.235,80.021,437.573,175.013,19.498,153.115
C08607=1087.230,79.743,437.592,175.011,19.496,153.115
C08608=1087.223,79.466,437.612,175.008,19.494,153.115
C08609=1087.217,79.188,437.630,175.006,19.492,153.115
C08610=1087.211,78.910,437.650,175.004,19.489,153.115
C08611=1087.205,78.661,437.667,175.002,19.488,153.115
C08612=1087.199,78.412,437.684,175.000,19.486,153.115
C08613=1087.194,78.162,437.701,174.999,19.484,153.115
C08614=1087.188,77.912,437.719,174.996,19.482,153.115
C08615=1087.182,77.663,437.737,174.995,19.480,153.115
C08616=1087.176,77.414,437.753,174.993,19.478,153.115
C08617=1087.171,77.165,437.770,174.991,19.477,153.115
C08618=1087.166,76.915,437.787,174.989,19.475,153.115
C08619=1087.159,76.667,437.804,174.987,19.473,153.115
C08620=1087.154,76.416,437.821,174.985,19.471,153.115
C08621=1087.148,76.167,437.839,174.984,19.470,153.114
C08622=1087.142,75.918,437.856,174.981,19.468,153.114
C08623=1087.137,75.669,437.873,174.980,19.466,153.114
C08624=1087.131,75.420,437.890,174.978,19.464,153.114
C08625=1087.126,75.170,437.907,174.976,19.463,153.114
C08626=1087.119,74.921,437.925,174.974,19.461,153.114
C08627=1087.114,74.671,437.941,174.972,19.459,153.114
C08628=1087.108,74.422,437.959,174.970,19.457,153.114
C08629=1087.102,74.173,437.975,174.969,19.456,153.114
C08630=1087.097,73.924,437.993,174.966,19.454,153.114
C08631=1087.092,73.674,438.010,174.965,19.452,153.114
C08632=1087.086,73.425,438.026,174.962,19.450,153.114
C08633=1087.080,73.176,438.043,174.961,19.449,153.114
C08634=1087.074,72.925,438.060,174.959,19.447,153.114
C08635=1087.068,72.676,438.078,174.957,19.445,153.114
C08636=1087.063,72.427,438.094,174.955,19.443,153.114
C08637=1087.057,72.178,438.111,174.954,19.442,153.114
C08638=1087.051,71.928,438.128,174.951,19.439,153.114
C08639=1087.046,71.679,438.145,174.950,19.438,153.114
C08640=1087.040,71.430,438.162,174.948,19.436,153.114
C08641=1087.035,71.180,438.179,174.946,19.434,153.114
C08642=1087.029,70.931,438.195,174.944,19.432,153.114
C08643=1087.023,70.682,438.213,174.942,19.431,153.114
C08644=1087.018,70.432,438.230,174.940,19.429,153.114
C08645=1087.011,70.183,438.247,174.939,19.427,153.114
C08646=1087.006,69.933,438.264,174.936,19.425,153.114
C08647=1087.000,69.684,438.280,174.935,19.423,153.113
C08648=1086.995,69.434,438.297,174.934,19.422,153.113
C08649=1086.989,69.185,438.314,174.931,19.420,153.113
C08650=1086.983,68.936,438.331,174.930,19.418,153.113
C08651=1086.977,68.686,438.347,174.928,19.416,153.113
C08652=1086.972,68.437,438.365,174.926,19.415,153.113
C08653=1086.966,68.188,438.381,174.924,19.413,153.113
C08654=1086.961,67.938,438.398,174.922,19.411,153.113
C08655=1086.955,67.689,438.414,174.920,19.409,153.113
C08656=1086.949,67.440,438.432,174.919,19.407,153.113
C08657=1086.943,67.191,438.448,174.917,19.405,153.113
C08658=1086.938,66.941,438.465,174.915,19.403,153.113
C08659=1086.932,66.692,438.481,174.913,19.401,153.113
C08660=1086.927,66.443,438.498,174.911,19.400,153.113
C08661=1086.921,66.193,438.515,174.909,19.398,153.113
C08662=1086.915,65.944,438.531,174.908,19.396,153.113
C08663=1086.910,65.694,438.548,174.906,19.394,153.113
C08664=1086.904,65.445,438.564,174.904,19.392,153.113
C08665=1086.898,65.196,438.582,174.902,19.390,153.113
C08666=1086.892,64.947,438.598,174.900,19.389,153.113
C08667=1086.887,64.697,438.615,174.899,19.387,153.113
C08668=1086.881,64.448,438.631,174.897,19.385,153.113
C08669=1086.874,64.197,438.648,174.895,19.384,153.113
C08670=1086.869,63.948,438.664,174.893,19.381,153.112
C08671=1086.862,63.671,438.682,174.891,19.379,153.112
C08672=1086.856,63.393,438.701,174.889,19.378,153.112
C08673=1086.849,63.115,438.720,174.887,19.376,153.112
C08674=1086.843,62.837,438.737,174.885,19.374,153.112
C08675=1086.837,62.587,438.754,174.884,19.372,153.112
C08676=1086.831,62.339,438.771,174.881,19.370,153.112
C08677=1086.826,62.089,438.787,174.880,19.368,153.112
C08678=1086.820,61.840,438.804,174.877,19.366,153.112
C08679=1086.814,61.590,438.820,174.876,19.365,153.112
C08680=1086.808,61.341,438.836,174.875,19.363,153.112
C08681=1086.803,61.091,438.853,174.872,19.361,153.112
C08682=1086.797,60.842,438.869,174.871,19.359,153.112
C08683=1086.791,60.593,438.886,174.869,19.357,153.112
C08684=1086.785,60.343,438.902,174.867,19.356,153.112
C08685=1086.779,60.094,438.918,174.865,19.353,153.112
C08686=1086.774,59.844,438.935,174.864,19.352,153.112
C08687=1086.768,59.595,438.951,174.861,19.350,153.112
C08688=1086.762,59.346,438.967,174.860,19.348,153.112
C08689=1086.756,59.096,438.984,174.858,19.346,153.112
C08690=1086.750,58.847,439.000,174.856,19.344,153.111
C08691=1086.745,58.597,439.017,174.855,19.343,153.111
C08692=1086.739,58.348,439.033,174.853,19.341,153.111
C08693=1086.733,58.099,439.049,174.851,19.339,153.111
C08694=1086.727,57.849,439.066,174.849,19.337,153.111
C08695=1086.721,57.599,439.081,174.848,19.335,153.111
C08696=1086.715,57.350,439.097,174.845,19.333,153.111
C08697=1086.710,57.100,439.114,174.844,19.332,153.111
C08698=1086.704,56.851,439.131,174.843,19.330,153.111
C08699=1086.698,56.602,439.147,174.840,19.328,153.111
C08700=1086.693,56.353,439.163,174.839,19.326,153.111
C08701=1086.687,56.104,439.179,174.837,19.324,153.111
C08702=1086.681,55.854,439.195,174.835,19.322,153.111
C08703=1086.675,55.605,439.211,174.833,19.320,153.111
C08704=1086.670,55.355,439.228,174.832,19.319,153.111
C08705=1086.664,55.105,439.244,174.829,19.317,153.111
C08706=1086.658,54.856,439.260,174.828,19.315,153.110
C08707=1086.652,54.607,439.276,174.827,19.313,153.110
C08708=1086.646,54.357,439.293,174.824,19.311,153.110
C08709=1086.641,54.108,439.308,174.823,19.310,153.110
C08710=1086.635,53.859,439.324,174.821,19.307,153.110
C08711=1086.629,53.609,439.340,174.819,19.306,153.110
C08712=1086.624,53.360,439.357,174.817,19.303,153.110
C08713=1086.618,53.110,439.373,174.816,19.302,153.110
C08714=1086.613,52.860,439.389,174.814,19.300,153.110
C08715=1086.607,52.611,439.405,174.812,19.298,153.110
C08716=1086.601,52.362,439.421,174.811,19.296,153.110
C08717=1086.595,52.113,439.437,174.809,19.294,153.110
C08718=1086.590,51.863,439.453,174.807,19.292,153.110
C08719=1086.584,51.614,439.469,174.806,19.291,153.110
C08720=1086.578,51.364,439.485,174.804,19.288,153.110
C08721=1086.573,51.115,439.501,174.802,19.287,153.109
C08722=1086.567,50.866,439.517,174.800,19.285,153.109
C08723=1086.562,50.616,439.534,174.799,19.283,153.109
C08724=1086.556,50.367,439.550,174.796,19.281,153.109
C08725=1086.550,50.117,439.565,174.795,19.279,153.109
C08726=1086.545,49.868,439.581,174.794,19.277,153.109
C08727=1086.539,49.619,439.598,174.791,19.275,153.109
C08728=1086.533,49.369,439.613,174.790,19.274,153.109
C08729=1086.527,49.119,439.629,174.788,19.271,153.109
C08730=1086.522,48.870,439.645,174.786,19.270,153.109
C08731=1086.516,48.621,439.661,174.784,19.268,153.109
C08732=1086.510,48.371,439.677,174.783,19.266,153.109
C08733=1086.504,48.121,439.693,174.782,19.264,153.109
C08734=1086.499,47.873,439.709,174.779,19.261,153.108
C08735=1086.493,47.594,439.727,174.778,19.260,153.108
C08736=1086.486,47.316,439.744,174.776,19.257,153.108
C08737=1086.480,47.038,439.762,174.774,19.255,153.108
C08738=1086.474,46.760,439.779,174.772,19.253,153.108
C08739=1086.468,46.511,439.796,174.770,19.251,153.108
C08740=1086.463,46.261,439.811,174.769,19.249,153.108
C08741=1086.457,46.012,439.827,174.767,19.247,153.108
C08742=1086.452,45.762,439.843,174.765,19.246,153.108
C08743=1086.446,45.513,439.859,174.763,19.243,153.108
C08744=1086.440,45.263,439.874,174.762,19.242,153.108
C08745=1086.435,45.014,439.890,174.760,19.240,153.107
C08746=1086.429,44.764,439.906,174.758,19.238,153.107
C08747=1086.423,44.515,439.922,174.757,19.236,153.107
C08748=1086.418,44.265,439.937,174.755,19.234,153.107
C08749=1086.412,44.016,439.953,174.753,19.232,153.107
C08750=1086.406,43.766,439.969,174.752,19.230,153.107
C08751=1086.401,43.517,439.985,174.750,19.228,153.107
C08752=1086.395,43.268,440.000,174.749,19.226,153.107
C08753=1086.389,43.018,440.016,174.746,19.224,153.107
C08754=1086.384,42.769,440.031,174.745,19.222,153.107
C08755=1086.378,42.519,440.047,174.744,19.220,153.107
C08756=1086.372,42.270,440.063,174.741,19.218,153.107
C08757=1086.366,42.020,440.078,174.740,19.216,153.106
C08758=1086.360,41.772,440.094,174.738,19.214,153.106
C08759=1086.355,41.522,440.109,174.736,19.213,153.106
C08760=1086.349,41.272,440.125,174.735,19.211,153.106
C08761=1086.344,41.023,440.141,174.733,19.209,153.106
C08762=1086.337,40.773,440.156,174.731,19.207,153.106
C08763=1086.332,40.523,440.171,174.730,19.205,153.106
C08764=1086.326,40.275,440.187,174.728,19.203,153.106
C08765=1086.321,40.025,440.203,174.727,19.201,153.106
C08766=1086.315,39.775,440.219,174.724,19.199,153.106
C08767=1086.309,39.526,440.234,174.723,19.197,153.106
C08768=1086.303,39.276,440.249,174.722,19.196,153.105
C08769=1086.298,39.026,440.265,174.719,19.194,153.106
C08770=1086.292,38.778,440.281,174.718,19.192,153.105
C08771=1086.286,38.528,440.296,174.716,19.190,153.105
C08772=1086.280,38.278,440.311,174.715,19.188,153.105
C08773=1086.275,38.030,440.327,174.713,19.186,153.105
C08774=1086.269,37.780,440.342,174.711,19.183,153.105
C08775=1086.263,37.530,440.357,174.710,19.182,153.105
C08776=1086.258,37.281,440.373,174.708,19.180,153.105
C08777=1086.252,37.031,440.389,174.706,19.178,153.105
C08778=1086.245,36.782,440.404,174.705,19.176,153.105
C08779=1086.240,36.532,440.419,174.703,19.174,153.105
C08780=1086.234,36.283,440.434,174.701,19.172,153.104
C08781=1086.229,36.034,440.450,174.700,19.171,153.104
C08782=1086.223,35.784,440.465,174.698,19.168,153.104
C08783=1086.217,35.534,440.480,174.696,19.167,153.104
C08784=1086.212,35.285,440.495,174.695,19.165,153.104
C08785=1086.205,35.036,440.510,174.693,19.163,153.104
C08786=1086.199,34.786,440.527,174.691,19.161,153.104
C08787=1086.194,34.537,440.542,174.690,19.159,153.104
C08788=1086.188,34.287,440.557,174.688,19.157,153.104
C08789=1086.183,34.038,440.572,174.687,19.156,153.104
C08790=1086.176,33.788,440.587,174.684,19.153,153.104
C08791=1086.171,33.538,440.602,174.683,19.151,153.104
C08792=1086.165,33.289,440.617,174.682,19.149,153.103
C08793=1086.159,33.040,440.633,174.680,19.147,153.103
C08794=1086.154,32.791,440.648,174.678,19.145,153.103
C08795=1086.148,32.541,440.663,174.677,19.144,153.103
C08796=1086.142,32.291,440.679,174.675,19.142,153.103
C08797=1086.136,32.042,440.694,174.673,19.140,153.103
C08798=1086.131,31.792,440.709,174.672,19.138,153.103
C08799=1086.124,31.514,440.726,174.670,19.136,153.103
C08800=1086.118,31.236,440.743,174.668,19.133,153.103
C08801=1086.111,30.958,440.760,174.666,19.132,153.103
C08802=1086.105,30.680,440.776,174.664,19.129,153.102
C08803=1086.100,30.431,440.791,174.663,19.128,153.102
C08804=1086.093,30.181,440.806,174.661,19.125,153.102
C08805=1086.088,29.932,440.822,174.659,19.124,153.102
C08806=1086.082,29.682,440.837,174.658,19.122,153.102
C08807=1086.077,29.433,440.852,174.656,19.120,153.102
C08808=1086.070,29.183,440.867,174.655,19.117,153.102
C08809=1086.065,28.934,440.882,174.653,19.116,153.102
C08810=1086.059,28.684,440.897,174.651,19.113,153.102
C08811=1086.054,28.435,440.912,174.650,19.112,153.102
C08812=1086.047,28.185,440.927,174.648,19.110,153.102
C08813=1086.042,27.936,440.942,174.646,19.108,153.101
C08814=1086.036,27.686,440.957,174.645,19.106,153.101
C08815=1086.030,27.437,440.972,174.643,19.104,153.101
C08816=1086.025,27.187,440.987,174.641,19.102,153.101
C08817=1086.019,26.938,441.002,174.640,19.100,153.101
C08818=1086.013,26.688,441.017,174.638,19.098,153.101
C08819=1086.007,26.439,441.032,174.637,19.096,153.101
C08820=1086.001,26.190,441.047,174.635,19.095,153.101
C08821=1085.995,25.940,441.062,174.633,19.093,153.101
C08822=1085.990,25.691,441.077,174.632,19.091,153.101
C08823=1085.983,25.441,441.091,174.630,19.089,153.101
C08824=1085.978,25.191,441.106,174.628,19.086,153.100
C08825=1085.972,24.942,441.121,174.627,19.085,153.100
C08826=1085.966,24.693,441.136,174.626,19.083,153.100
C08827=1085.961,24.443,441.151,174.623,19.081,153.100
C08828=1085.955,24.194,441.166,174.622,19.079,153.100
C08829=1085.948,23.944,441.181,174.621,19.077,153.100
C08830=1085.944,23.694,441.195,174.619,19.075,153.100
C08831=1085.938,23.445,441.210,174.617,19.073,153.100
C08832=1085.932,23.196,441.225,174.616,19.072,153.100
C08833=1085.927,22.946,441.240,174.614,19.069,153.100
C08834=1085.920,22.697,441.255,174.612,19.068,153.100
C08835=1085.915,22.447,441.269,174.611,19.066,153.099
C08836=1085.908,22.197,441.284,174.609,19.064,153.099
C08837=1085.903,21.948,441.299,174.608,19.062,153.099
C08838=1085.897,21.699,441.314,174.606,19.060,153.099
C08839=1085.891,21.450,441.328,174.604,19.057,153.099
C08840=1085.886,21.199,441.343,174.603,19.056,153.099
C08841=1085.880,20.950,441.358,174.601,19.054,153.099
C08842=1085.874,20.701,441.372,174.599,19.052,153.099
C08843=1085.868,20.451,441.387,174.598,19.050,153.099
C08844=1085.863,20.202,441.402,174.597,19.048,153.099
C08845=1085.857,19.952,441.417,174.595,19.046,153.098
C08846=1085.851,19.703,441.431,174.593,19.044,153.098
C08847=1085.845,19.453,441.446,174.592,19.042,153.098
C08848=1085.839,19.204,441.460,174.590,19.041,153.098
C08849=1085.834,18.954,441.475,174.588,19.038,153.098
C08850=1085.828,18.704,441.490,174.587,19.037,153.098
C08851=1085.822,18.455,441.504,174.586,19.035,153.098
C08852=1085.816,18.206,441.519,174.583,19.033,153.098
C08853=1085.810,17.956,441.533,174.582,19.030,153.098
C08854=1085.804,17.707,441.548,174.581,19.029,153.098
C08855=1085.799,17.457,441.563,174.579,19.026,153.097
C08856=1085.793,17.207,441.577,174.577,19.025,153.097
C08857=1085.787,16.958,441.592,174.576,19.023,153.097
C08858=1085.781,16.708,441.606,174.574,19.021,153.097
C08859=1085.776,16.459,441.620,174.573,19.019,153.097
C08860=1085.769,16.210,441.635,174.571,19.017,153.097
C08861=1085.765,15.960,441.650,174.569,19.015,153.097
C08862=1085.759,15.711,441.664,174.568,19.013,153.097
C08863=1085.752,15.434,441.681,174.567,19.011,153.097
C08864=1085.746,15.157,441.696,174.564,19.009,153.097
C08865=1085.739,14.881,441.712,174.562,19.007,153.096
C08866=1085.733,14.604,441.728,174.561,19.005,153.096
C08867=1085.727,14.355,441.743,174.560,19.003,153.096
C08868=1085.721,14.105,441.757,174.558,19.000,153.096
C08869=1085.715,13.856,441.771,174.556,18.999,153.096
C08870=1085.709,13.605,441.786,174.555,18.997,153.096
C08871=1085.703,13.356,441.800,174.553,18.995,153.096
C08872=1085.698,13.107,441.814,174.551,18.993,153.096
C08873=1085.691,12.857,441.829,174.550,18.991,153.096
C08874=1085.686,12.608,441.843,174.549,18.990,153.096
C08875=1085.680,12.359,441.858,174.546,18.987,153.095
C08876=1085.674,12.108,441.872,174.545,18.986,153.095
C08877=1085.668,11.859,441.886,174.544,18.984,153.095
C08878=1085.662,11.609,441.901,174.542,18.982,153.095
C08879=1085.656,11.360,441.915,174.540,18.980,153.095
C08880=1085.651,11.111,441.929,174.539,18.978,153.095
C08881=1085.645,10.860,441.943,174.537,18.976,153.095
C08882=1085.639,10.611,441.958,174.535,18.974,153.095
C08883=1085.633,10.362,441.972,174.534,18.972,153.095
C08884=1085.627,10.112,441.987,174.533,18.970,153.095
C08885=1085.622,9.863,442.000,174.531,18.968,153.095
C08886=1085.615,9.614,442.014,174.529,18.966,153.094
C08887=1085.609,9.364,442.029,174.528,18.965,153.094
C08888=1085.603,9.114,442.043,174.526,18.962,153.094
C08889=1085.598,8.865,442.057,174.524,18.961,153.094
C08890=1085.592,8.615,442.071,174.523,18.959,153.094
C08891=1085.586,8.365,442.085,174.522,18.957,153.094
C08892=1085.580,8.116,442.100,174.520,18.955,153.094
C08893=1085.575,7.867,442.114,174.518,18.953,153.094
C08894=1085.569,7.616,442.128,174.517,18.951,153.094
C08895=1085.563,7.367,442.142,174.515,18.949,153.094
C08896=1085.557,7.118,442.156,174.513,18.947,153.094
C08897=1085.551,6.868,442.170,174.512,18.945,153.093
C08898=1085.545,6.619,442.185,174.511,18.944,153.093
C08899=1085.539,6.369,442.198,174.509,18.941,153.093
C08900=1085.534,6.120,442.212,174.507,18.940,153.093
C08901=1085.528,5.870,442.227,174.506,18.938,153.093
C08902=1085.522,5.621,442.241,174.505,18.936,153.093
C08903=1085.516,5.371,442.254,174.503,18.934,153.093
C08904=1085.510,5.122,442.268,174.501,18.932,153.093
C08905=1085.504,4.872,442.283,174.500,18.930,153.093
C08906=1085.499,4.622,442.297,174.498,18.928,153.093
C08907=1085.493,4.373,442.311,174.497,18.926,153.092
C08908=1085.488,4.123,442.325,174.495,18.924,153.092
C08909=1085.482,3.874,442.339,174.494,18.922,153.092
C08910=1085.475,3.624,442.353,174.492,18.920,153.092
C08911=1085.470,3.375,442.367,174.490,18.918,153.092
C08912=1085.464,3.125,442.381,174.489,18.917,153.092
C08913=1085.459,2.876,442.395,174.487,18.914,153.092
C08914=1085.453,2.626,442.408,174.486,18.913,153.092
C08915=1085.447,2.376,442.423,174.484,18.911,153.092
C08916=1085.441,2.127,442.437,174.483,18.909,153.091
C08917=1085.435,1.878,442.451,174.481,18.907,153.091
C08918=1085.430,1.628,442.464,174.479,18.905,153.091
C08919=1085.424,1.378,442.478,174.478,18.903,153.091
C08920=1085.418,1.128,442.492,174.477,18.901,153.091
C08921=1085.412,0.879,442.506,174.475,18.899,153.091
C08922=1085.406,0.630,442.520,174.473,18.897,153.091
C08923=1085.401,0.380,442.534,174.472,18.895,153.091
C08924=1085.395,0.131,442.548,174.471,18.894,153.091
C08925=1085.390,-0.119,442.562,174.469,18.891,153.091
C08926=1085.383,-0.368,442.575,174.467,18.889,153.090
C08927=1085.377,-0.643,442.590,174.466,18.888,153.090
C08928=1085.371,-0.918,442.606,174.464,18.885,153.090
C08929=1085.365,-1.193,442.621,174.463,18.883,153.090
C08930=1085.358,-1.467,442.637,174.461,18.881,153.090
C08931=1085.353,-1.717,442.651,174.459,18.879,153.090
C08932=1085.347,-1.966,442.664,174.458,18.877,153.090
C08933=1085.341,-2.216,442.678,174.456,18.875,153.090
C08934=1085.336,-2.465,442.692,174.454,18.873,153.090
C08935=1085.330,-2.715,442.705,174.453,18.871,153.089
C08936=1085.323,-2.965,442.719,174.451,18.869,153.089
C08937=1085.318,-3.214,442.733,174.450,18.867,153.089
C08938=1085.312,-3.464,442.747,174.448,18.866,153.089
C08939=1085.306,-3.713,442.760,174.447,18.864,153.089
C08940=1085.301,-3.963,442.774,174.445,18.862,153.089
C08941=1085.294,-4.212,442.787,174.444,18.860,153.089
C08942=1085.289,-4.462,442.801,174.442,18.858,153.089
C08943=1085.283,-4.712,442.815,174.441,18.856,153.089
C08944=1085.277,-4.961,442.829,174.439,18.854,153.089
C08945=1085.271,-5.211,442.842,174.438,18.852,153.088
C08946=1085.265,-5.460,442.856,174.436,18.850,153.088
C08947=1085.259,-5.710,442.870,174.435,18.849,153.088
C08948=1085.253,-5.959,442.883,174.434,18.847,153.088
C08949=1085.248,-6.209,442.896,174.431,18.845,153.088
C08950=1085.241,-6.459,442.910,174.430,18.843,153.088
C08951=1085.236,-6.709,442.923,174.429,18.841,153.088
C08952=1085.230,-6.958,442.937,174.427,18.839,153.088
C08953=1085.224,-7.207,442.951,174.425,18.837,153.088
C08954=1085.218,-7.457,442.964,174.424,18.836,153.088
C08955=1085.212,-7.706,442.978,174.423,18.833,153.088
C08956=1085.206,-7.955,442.991,174.421,18.832,153.087
C08957=1085.201,-8.205,443.005,174.419,18.829,153.087
C08958=1085.195,-8.455,443.017,174.418,18.828,153.087
C08959=1085.189,-8.704,443.031,174.416,18.826,153.087
C08960=1085.183,-8.954,443.045,174.415,18.824,153.087
C08961=1085.177,-9.204,443.059,174.413,18.822,153.087
C08962=1085.171,-9.453,443.072,174.412,18.820,153.087
C08963=1085.165,-9.703,443.086,174.410,18.819,153.087
C08964=1085.159,-9.953,443.098,174.409,18.817,153.087
C08965=1085.154,-10.202,443.112,174.407,18.815,153.087
C08966=1085.148,-10.452,443.126,174.406,18.812,153.086
C08967=1085.142,-10.701,443.139,174.404,18.811,153.086
C08968=1085.136,-10.951,443.152,174.403,18.809,153.086
C08969=1085.131,-11.201,443.166,174.401,18.807,153.086
C08970=1085.125,-11.450,443.179,174.399,18.805,153.086
C08971=1085.118,-11.699,443.192,174.398,18.803,153.086
C08972=1085.113,-11.949,443.206,174.397,18.801,153.086
C08973=1085.107,-12.199,443.219,174.395,18.800,153.086
C08974=1085.102,-12.448,443.233,174.393,18.798,153.086
C08975=1085.095,-12.697,443.246,174.392,18.796,153.086
C08976=1085.090,-12.948,443.259,174.390,18.794,153.086
C08977=1085.084,-13.197,443.272,174.389,18.792,153.085
C08978=1085.078,-13.446,443.286,174.388,18.790,153.085
C08979=1085.072,-13.696,443.300,174.386,18.788,153.085
C08980=1085.066,-13.946,443.312,174.384,18.786,153.085
C08981=1085.061,-14.195,443.326,174.383,18.784,153.085
C08982=1085.055,-14.444,443.339,174.382,18.783,153.085
C08983=1085.050,-14.695,443.352,174.380,18.780,153.085
C08984=1085.043,-14.944,443.366,174.378,18.779,153.085
C08985=1085.037,-15.193,443.379,174.377,18.777,153.085
C08986=1085.032,-15.443,443.392,174.376,18.775,153.085
C08987=1085.026,-15.693,443.405,174.374,18.774,153.085
C08988=1085.020,-15.943,443.418,174.372,18.771,153.084
C08989=1085.014,-16.192,443.431,174.371,18.769,153.084
C08990=1085.008,-16.441,443.445,174.369,18.768,153.084
C08991=1085.001,-16.715,443.460,174.367,18.765,153.084
C08992=1084.995,-16.987,443.474,174.366,18.764,153.084
C08993=1084.989,-17.261,443.488,174.365,18.762,153.084
C08994=1084.983,-17.534,443.502,174.362,18.760,153.084
C08995=1084.976,-17.783,443.515,174.361,18.758,153.084
C08996=1084.970,-18.033,443.529,174.360,18.756,153.084
C08997=1084.964,-18.283,443.541,174.359,18.754,153.084
C08998=1084.958,-18.532,443.554,174.356,18.752,153.084
C08999=1084.953,-18.782,443.568,174.355,18.751,153.084
C09000=1084.947,-19.031,443.581,174.354,18.748,153.083
C09001=1084.941,-19.281,443.593,174.352,18.747,153.083
C09002=1084.934,-19.530,443.607,174.351,18.745,153.083
C09003=1084.929,-19.781,443.620,174.349,18.743,153.083
C09004=1084.923,-20.030,443.633,174.347,18.741,153.083
C09005=1084.917,-20.280,443.646,174.346,18.739,153.083
C09006=1084.911,-20.529,443.659,174.345,18.738,153.083
C09007=1084.905,-20.779,443.671,174.343,18.736,153.083
C09008=1084.900,-21.028,443.685,174.341,18.734,153.083
C09009=1084.894,-21.278,443.697,174.340,18.732,153.083
C09010=1084.888,-21.527,443.711,174.339,18.731,153.083
C09011=1084.882,-21.777,443.723,174.337,18.728,153.082
C09012=1084.876,-22.026,443.737,174.336,18.727,153.082
C09013=1084.871,-22.276,443.750,174.334,18.724,153.082
C09014=1084.865,-22.525,443.763,174.332,18.723,153.082
C09015=1084.859,-22.775,443.776,174.331,18.721,153.082
C09016=1084.853,-23.025,443.788,174.330,18.719,153.082
C09017=1084.847,-23.275,443.801,174.328,18.718,153.082
C09018=1084.841,-23.524,443.814,174.326,18.715,153.082
C09019=1084.836,-23.773,443.827,174.325,18.714,153.082
C09020=1084.830,-24.023,443.840,174.324,18.712,153.082
C09021=1084.824,-24.273,443.853,174.322,18.710,153.082
C09022=1084.818,-24.522,443.866,174.321,18.708,153.082
C09023=1084.812,-24.772,443.878,174.319,18.707,153.081
C09024=1084.806,-25.021,443.892,174.317,18.704,153.081
C09025=1084.800,-25.271,443.904,174.316,18.703,153.081
C09026=1084.795,-25.522,443.917,174.315,18.701,153.081
C09027=1084.789,-25.770,443.930,174.313,18.699,153.081
C09028=1084.783,-26.020,443.943,174.312,18.698,153.081
C09029=1084.777,-26.270,443.955,174.310,18.695,153.081
C09030=1084.771,-26.519,443.969,174.309,18.694,153.081
C09031=1084.765,-26.769,443.981,174.307,18.692,153.081
C09032=1084.759,-27.019,443.994,174.306,18.690,153.081
C09033=1084.754,-27.268,444.006,174.304,18.688,153.081
C09034=1084.748,-27.517,444.019,174.303,18.687,153.081
C09035=1084.742,-27.767,444.032,174.301,18.684,153.080
C09036=1084.736,-28.017,444.044,174.300,18.683,153.080
C09037=1084.729,-28.266,444.058,174.298,18.681,153.080
C09038=1084.724,-28.516,444.070,174.297,18.679,153.080
C09039=1084.718,-28.766,444.083,174.296,18.678,153.080
C09040=1084.712,-29.016,444.095,174.293,18.676,153.080
C09041=1084.706,-29.265,444.108,174.292,18.674,153.080
C09042=1084.700,-29.514,444.121,174.291,18.672,153.080
C09043=1084.694,-29.764,444.133,174.289,18.671,153.080
C09044=1084.688,-30.014,444.146,174.288,18.669,153.080
C09045=1084.682,-30.263,444.159,174.287,18.667,153.080
C09046=1084.676,-30.513,444.172,174.284,18.665,153.080
C09047=1084.670,-30.762,444.183,174.283,18.663,153.080
C09048=1084.664,-31.012,444.196,174.282,18.662,153.080
C09049=1084.658,-31.262,444.208,174.280,18.660,153.079
C09050=1084.652,-31.511,444.222,174.279,18.658,153.079
C09051=1084.646,-31.761,444.234,174.277,18.657,153.079
C09052=1084.640,-32.011,444.247,174.275,18.654,153.079
C09053=1084.635,-32.260,444.259,174.274,18.653,153.079
C09054=1084.629,-32.510,444.271,174.273,18.651,153.079
C09055=1084.622,-32.782,444.285,174.271,18.649,153.079
C09056=1084.617,-33.054,444.299,174.269,18.647,153.079
C09057=1084.610,-33.327,444.313,174.268,18.645,153.079
C09058=1084.603,-33.599,444.326,174.267,18.643,153.079
C09059=1084.598,-33.848,444.338,174.265,18.642,153.079
C09060=1084.592,-34.098,444.351,174.263,18.640,153.079
C09061=1084.586,-34.348,444.364,174.262,18.638,153.079
C09062=1084.580,-34.598,444.376,174.260,18.636,153.078
C09063=1084.575,-34.847,444.388,174.259,18.635,153.078
C09064=1084.568,-35.097,444.400,174.257,18.633,153.078
C09065=1084.562,-35.346,444.414,174.256,18.631,153.078
C09066=1084.556,-35.596,444.426,174.255,18.629,153.078
C09067=1084.550,-35.845,444.438,174.253,18.627,153.078
C09068=1084.545,-36.095,444.451,174.251,18.626,153.078
C09069=1084.539,-36.345,444.463,174.250,18.624,153.078
C09070=1084.533,-36.595,444.476,174.248,18.622,153.078
C09071=1084.527,-36.844,444.488,174.247,18.621,153.078
C09072=1084.521,-37.093,444.500,174.246,18.619,153.078
C09073=1084.515,-37.343,444.513,174.244,18.617,153.078
C09074=1084.510,-37.592,444.525,174.242,18.615,153.078
C09075=1084.504,-37.842,444.537,174.241,18.614,153.078
C09076=1084.498,-38.092,444.550,174.240,18.611,153.077
C09077=1084.492,-38.342,444.562,174.238,18.610,153.077
C09078=1084.486,-38.591,444.574,174.237,18.608,153.077
C09079=1084.480,-38.841,444.587,174.235,18.607,153.077
C09080=1084.474,-39.091,444.599,174.234,18.605,153.077
C09081=1084.469,-39.340,444.611,174.232,18.603,153.077
C09082=1084.462,-39.590,444.623,174.230,18.601,153.077
C09083=1084.456,-39.839,444.636,174.229,18.600,153.077
C09084=1084.450,-40.089,444.648,174.228,18.598,153.077
C09085=1084.444,-40.339,444.659,174.226,18.597,153.077
C09086=1084.439,-40.589,444.672,174.225,18.595,153.077
C09087=1084.433,-40.839,444.684,174.224,18.593,153.077
C09088=1084.426,-41.088,444.696,174.221,18.591,153.077
C09089=1084.421,-41.337,444.709,174.220,18.589,153.077
C09090=1084.415,-41.587,444.721,174.218,18.588,153.077
C09091=1084.408,-41.837,444.733,174.217,18.586,153.077
C09092=1084.403,-42.086,444.745,174.216,18.585,153.077
C09093=1084.396,-42.336,444.757,174.214,18.583,153.077
C09094=1084.390,-42.585,444.770,174.213,18.581,153.076
C09095=1084.385,-42.835,444.781,174.212,18.580,153.076
C09096=1084.379,-43.085,444.793,174.209,18.578,153.076
C09097=1084.373,-43.335,444.806,174.208,18.576,153.076
C09098=1084.367,-43.584,444.818,174.206,18.574,153.076
C09099=1084.361,-43.833,444.830,174.205,18.572,153.076
C09100=1084.355,-44.083,444.842,174.204,18.571,153.076
C09101=1084.349,-44.333,444.853,174.202,18.569,153.076
C09102=1084.343,-44.583,444.866,174.201,18.568,153.076
C09103=1084.337,-44.833,444.878,174.200,18.566,153.076
C09104=1084.331,-45.081,444.890,174.198,18.565,153.076
C09105=1084.325,-45.331,444.903,174.196,18.563,153.076
